LIN {X 0,Y 573.583,Z 173.358,A -85,B 0,C 180,E1 -2266.731,E2 -2266.731} C_VEL
LIN {X 0,Y 573.739,Z 153.891,A -85,B 0,C 180,E1 -2269.402,E2 -2269.402} C_VEL
LIN {X 0,Y 573.978,Z 134.192,A -85,B 0,C 180,E1 -2272.118,E2 -2272.118} C_VEL
LIN {X 0,Y 573.92,Z 125.746,A -85,B 0,C 180,E1 -2273.303,E2 -2273.303} C_VEL
LIN {X 0,Y 573.25,Z 122.082,A -85,B 0,C 180,E1 -2273.864,E2 -2273.864} C_VEL
LIN {X 0,Y 573.237,Z 122.08,A -85,B 0,C 180,E1 -2276.492,E2 -2276.492} C_VEL
LIN {X 0,Y 573.262,Z 122.073,A -85,B 0,C 180,E1 -2279.366,E2 -2279.366} C_VEL
LIN {X 0,Y 573.25,Z 122.079,A -85,B 0,C 180,E1 -2282.227,E2 -2282.227} C_VEL
LIN {X 0,Y 573.235,Z 122.075,A -85,B 0,C 180,E1 -2284.771,E2 -2284.771} C_VEL
LIN {X 0,Y 573.236,Z 122.084,A -85,B 0,C 180,E1 -2287.807,E2 -2287.807} C_VEL
LIN {X 0,Y 573.246,Z 122.074,A -85,B 0,C 180,E1 -2290.525,E2 -2290.525} C_VEL
LIN {X 0,Y 573.237,Z 122.078,A -85,B 0,C 180,E1 -2293.359,E2 -2293.359} C_VEL
LIN {X 0,Y 573.246,Z 122.075,A -85,B 0,C 180,E1 -2296.331,E2 -2296.331} C_VEL
LIN {X 0,Y 573.23,Z 122.075,A -85,B 0,C 180,E1 -2298.543,E2 -2298.543} C_VEL
LIN {X 0,Y 573.242,Z 122.079,A -85,B 0,C 180,E1 -2301.298,E2 -2301.298} C_VEL
LIN {X 0,Y 573.213,Z 122.08,A -85,B 0,C 180,E1 -2304.018,E2 -2304.018} C_VEL
LIN {X 0,Y 573.239,Z 122.074,A -85,B 0,C 180,E1 -2306.516,E2 -2306.516} C_VEL
LIN {X 0,Y 573.224,Z 122.081,A -85,B 0,C 180,E1 -2309.118,E2 -2309.118} C_VEL
LIN {X 0,Y 573.251,Z 122.074,A -85,B 0,C 180,E1 -2311.971,E2 -2311.971} C_VEL
LIN {X 0,Y 573.248,Z 122.074,A -85,B 0,C 180,E1 -2314.589,E2 -2314.589} C_VEL
LIN {X 0,Y 573.235,Z 122.078,A -85,B 0,C 180,E1 -2317.662,E2 -2317.662} C_VEL
LIN {X 0,Y 573.267,Z 122.074,A -85,B 0,C 180,E1 -2320.67,E2 -2320.67} C_VEL
LIN {X 0,Y 573.24,Z 122.076,A -85,B 0,C 180,E1 -2323.621,E2 -2323.621} C_VEL
LIN {X 0,Y 573.273,Z 122.07,A -85,B 0,C 180,E1 -2325.807,E2 -2325.807} C_VEL
LIN {X 0,Y 573.264,Z 122.078,A -85,B 0,C 180,E1 -2328.745,E2 -2328.745} C_VEL
LIN {X 0,Y 573.254,Z 122.073,A -85,B 0,C 180,E1 -2331.54,E2 -2331.54} C_VEL
LIN {X 0,Y 573.298,Z 122.07,A -85,B 0,C 180,E1 -2334.372,E2 -2334.372} C_VEL
LIN {X 0,Y 573.313,Z 122.065,A -85,B 0,C 180,E1 -2337.892,E2 -2337.892} C_VEL
LIN {X 0,Y 573.334,Z 122.072,A -85,B 0,C 180,E1 -2340.702,E2 -2340.702} C_VEL
LIN {X 0,Y 573.305,Z 122.073,A -85,B 0,C 180,E1 -2342.81,E2 -2342.81} C_VEL
LIN {X 0,Y 573.29,Z 122.068,A -85,B 0,C 180,E1 -2345.628,E2 -2345.628} C_VEL
LIN {X 0,Y 573.283,Z 122.078,A -85,B 0,C 180,E1 -2348.459,E2 -2348.459} C_VEL
LIN {X 0,Y 573.272,Z 122.07,A -85,B 0,C 180,E1 -2351.312,E2 -2351.312} C_VEL
LIN {X 0,Y 573.281,Z 122.078,A -85,B 0,C 180,E1 -2354.424,E2 -2354.424} C_VEL
LIN {X 0,Y 573.258,Z 122.072,A -85,B 0,C 180,E1 -2357.111,E2 -2357.111} C_VEL
LIN {X 0,Y 573.24,Z 122.081,A -85,B 0,C 180,E1 -2360.077,E2 -2360.077} C_VEL
LIN {X 0,Y 573.234,Z 122.082,A -85,B 0,C 180,E1 -2362.338,E2 -2362.338} C_VEL
LIN {X 0,Y 573.248,Z 122.075,A -85,B 0,C 180,E1 -2364.39,E2 -2364.39} C_VEL
LIN {X 0,Y 572.622,Z 122.155,A -85,B 0,C 180,E1 -2364.976,E2 -2364.976} C_VEL
LIN {X 0,Y 569.773,Z 122.513,A -85,B 0,C 180,E1 -2365.927,E2 -2365.927} C_VEL
LIN {X 0,Y 567.334,Z 122.813,A -85,B 0,C 180,E1 -2366.693,E2 -2366.693} C_VEL
LIN {X 0,Y 566.275,Z 122.942,A -85,B 0,C 180,E1 -2367.284,E2 -2367.284} C_VEL
LIN {X 0,Y 566.184,Z 122.954,A -85,B 0,C 180,E1 -2367.484,E2 -2367.484} C_VEL
LIN {X 0,Y 566.199,Z 122.957,A -85,B 0,C 180,E1 -2369.769,E2 -2369.769} C_VEL
LIN {X 0,Y 566.201,Z 122.954,A -85,B 0,C 180,E1 -2372.43,E2 -2372.43} C_VEL
LIN {X 0,Y 566.178,Z 122.954,A -85,B 0,C 180,E1 -2374.989,E2 -2374.989} C_VEL
LIN {X 0,Y 566.195,Z 122.956,A -85,B 0,C 180,E1 -2377.461,E2 -2377.461} C_VEL
LIN {X 0,Y 566.208,Z 122.953,A -85,B 0,C 180,E1 -2380.199,E2 -2380.199} C_VEL
LIN {X 0,Y 566.199,Z 122.952,A -85,B 0,C 180,E1 -2383.054,E2 -2383.054} C_VEL
LIN {X 0,Y 566.197,Z 122.955,A -85,B 0,C 180,E1 -2386.049,E2 -2386.049} C_VEL
LIN {X 0,Y 566.203,Z 122.955,A -85,B 0,C 180,E1 -2389.215,E2 -2389.215} C_VEL
LIN {X 0,Y 566.184,Z 122.961,A -85,B 0,C 180,E1 -2391.637,E2 -2391.637} C_VEL
LIN {X 0,Y 566.161,Z 122.956,A -85,B 0,C 180,E1 -2394.308,E2 -2394.308} C_VEL
LIN {X 0,Y 566.203,Z 122.953,A -85,B 0,C 180,E1 -2396.897,E2 -2396.897} C_VEL
LIN {X 0,Y 566.174,Z 122.963,A -85,B 0,C 180,E1 -2399.407,E2 -2399.407} C_VEL
LIN {X 0,Y 566.194,Z 122.954,A -85,B 0,C 180,E1 -2401.857,E2 -2401.857} C_VEL
LIN {X 0,Y 566.209,Z 122.95,A -85,B 0,C 180,E1 -2404.251,E2 -2404.251} C_VEL
LIN {X 0,Y 566.168,Z 122.958,A -85,B 0,C 180,E1 -2406.72,E2 -2406.72} C_VEL
LIN {X 0,Y 566.205,Z 122.952,A -85,B 0,C 180,E1 -2409.663,E2 -2409.663} C_VEL
LIN {X 0,Y 566.196,Z 122.956,A -85,B 0,C 180,E1 -2412.668,E2 -2412.668} C_VEL
LIN {X 0,Y 566.221,Z 122.95,A -85,B 0,C 180,E1 -2415.627,E2 -2415.627} C_VEL
LIN {X 0,Y 566.235,Z 122.953,A -85,B 0,C 180,E1 -2418.676,E2 -2418.676} C_VEL
LIN {X 0,Y 566.205,Z 122.952,A -85,B 0,C 180,E1 -2421.434,E2 -2421.434} C_VEL
LIN {X 0,Y 566.265,Z 122.946,A -85,B 0,C 180,E1 -2424.302,E2 -2424.302} C_VEL
LIN {X 0,Y 566.283,Z 122.942,A -85,B 0,C 180,E1 -2427.866,E2 -2427.866} C_VEL
LIN {X 0,Y 566.303,Z 122.948,A -85,B 0,C 180,E1 -2430.711,E2 -2430.711} C_VEL
LIN {X 0,Y 566.274,Z 123.08,A -85,B 0,C 180,E1 -2431.6,E2 -2431.6} C_VEL
LIN {X 0,Y 566.359,Z 131.56,A -85,B 0,C 180,E1 -2433.201,E2 -2433.201} C_VEL
LIN {X 0,Y 566.17,Z 146.716,A -85,B 0,C 180,E1 -2436.057,E2 -2436.057} C_VEL
LIN {X 0,Y 567.134,Z 152.715,A -85,B 0,C 180,E1 -2436.158,E2 -2436.158} C_VEL
LIN {X 0,Y 566.874,Z 253.461,A -85,B 0,C 180,E1 -2437.456,E2 -2437.456} C_VEL
LIN {X 0,Y 566.817,Z 267.103,A -85,B 0,C 180,E1 -2437.79,E2 -2437.79} C_VEL
LIN {X 0,Y 566.718,Z 279.633,A -85,B 0,C 180,E1 -2438.244,E2 -2438.244} C_VEL
LIN {X 0,Y 566.604,Z 291.505,A -85,B 0,C 180,E1 -2438.83,E2 -2438.83} C_VEL
LIN {X 0,Y 566.448,Z 302.94,A -85,B 0,C 180,E1 -2439.552,E2 -2439.552} C_VEL
LIN {X 0,Y 566.305,Z 313.27,A -85,B 0,C 180,E1 -2440.367,E2 -2440.367} C_VEL
LIN {X 0,Y 566.179,Z 322.76,A -85,B 0,C 180,E1 -2441.296,E2 -2441.296} C_VEL
LIN {X 0,Y 566.072,Z 331.625,A -85,B 0,C 180,E1 -2442.367,E2 -2442.367} C_VEL
LIN {X 0,Y 566.022,Z 338.925,A -85,B 0,C 180,E1 -2443.463,E2 -2443.463} C_VEL
LIN {X 0,Y 565.955,Z 345.411,A -85,B 0,C 180,E1 -2444.711,E2 -2444.711} C_VEL
LIN {X 0,Y 565.893,Z 349.972,A -85,B 0,C 180,E1 -2445.856,E2 -2445.856} C_VEL
LIN {X 0,Y 565.855,Z 353.302,A -85,B 0,C 180,E1 -2446.991,E2 -2446.991} C_VEL
LIN {X 0,Y 565.837,Z 355.482,A -85,B 0,C 180,E1 -2448.09,E2 -2448.09} C_VEL
LIN {X 0,Y 565.872,Z 356.753,A -85,B 0,C 180,E1 -2449.283,E2 -2449.283} C_VEL
LIN {X 0,Y 565.836,Z 356.938,A -85,B 0,C 180,E1 -2450.351,E2 -2450.351} C_VEL
LIN {X 0,Y 565.864,Z 356.337,A -85,B 0,C 180,E1 -2451.331,E2 -2451.331} C_VEL
LIN {X 0,Y 565.858,Z 354.318,A -85,B 0,C 180,E1 -2452.645,E2 -2452.645} C_VEL
LIN {X 0,Y 565.904,Z 351.363,A -85,B 0,C 180,E1 -2453.805,E2 -2453.805} C_VEL
LIN {X 0,Y 565.924,Z 347.174,A -85,B 0,C 180,E1 -2454.976,E2 -2454.976} C_VEL
LIN {X 0,Y 565.99,Z 341.588,A -85,B 0,C 180,E1 -2456.156,E2 -2456.156} C_VEL
LIN {X 0,Y 566.049,Z 334.295,A -85,B 0,C 180,E1 -2457.348,E2 -2457.348} C_VEL
LIN {X 0,Y 566.132,Z 326.85,A -85,B 0,C 180,E1 -2458.329,E2 -2458.329} C_VEL
LIN {X 0,Y 566.255,Z 317.253,A -85,B 0,C 180,E1 -2459.357,E2 -2459.357} C_VEL
LIN {X 0,Y 566.365,Z 306.538,A -85,B 0,C 180,E1 -2460.273,E2 -2460.273} C_VEL
LIN {X 0,Y 566.505,Z 295.04,A -85,B 0,C 180,E1 -2461.058,E2 -2461.058} C_VEL
LIN {X 0,Y 566.696,Z 282.783,A -85,B 0,C 180,E1 -2461.704,E2 -2461.704} C_VEL
LIN {X 0,Y 566.826,Z 269.71,A -85,B 0,C 180,E1 -2462.219,E2 -2462.219} C_VEL
LIN {X 0,Y 566.924,Z 256.913,A -85,B 0,C 180,E1 -2462.564,E2 -2462.564} C_VEL
LIN {X 0,Y 566.964,Z 241.389,A -85,B 0,C 180,E1 -2462.805,E2 -2462.805} C_VEL
LIN {X 0,Y 567.146,Z 152.118,A -85,B 0,C 180,E1 -2463.939,E2 -2463.939} C_VEL
LIN {X 0,Y 566.206,Z 146.617,A -85,B 0,C 180,E1 -2464.047,E2 -2464.047} C_VEL
LIN {X 0,Y 566.359,Z 132.186,A -85,B 0,C 180,E1 -2466.776,E2 -2466.776} C_VEL
LIN {X 0,Y 566.237,Z 123.074,A -85,B 0,C 180,E1 -2468.463,E2 -2468.463} C_VEL
LIN {X 0,Y 566.166,Z 122.963,A -85,B 0,C 180,E1 -2471.141,E2 -2471.141} C_VEL
LIN {X 0,Y 566.158,Z 122.959,A -85,B 0,C 180,E1 -2474.04,E2 -2474.04} C_VEL
LIN {X 0,Y 566.182,Z 122.963,A -85,B 0,C 180,E1 -2477.085,E2 -2477.085} C_VEL
LIN {X 0,Y 566.205,Z 122.952,A -85,B 0,C 180,E1 -2479.801,E2 -2479.801} C_VEL
LIN {X 0,Y 566.192,Z 122.956,A -85,B 0,C 180,E1 -2482.6,E2 -2482.6} C_VEL
LIN {X 0,Y 566.182,Z 122.96,A -85,B 0,C 180,E1 -2485.18,E2 -2485.18} C_VEL
LIN {X 0,Y 566.217,Z 122.95,A -85,B 0,C 180,E1 -2487.743,E2 -2487.743} C_VEL
LIN {X 0,Y 566.149,Z 122.961,A -85,B 0,C 180,E1 -2490.338,E2 -2490.338} C_VEL
LIN {X 0,Y 566.175,Z 122.956,A -85,B 0,C 180,E1 -2493.457,E2 -2493.457} C_VEL
LIN {X 0,Y 566.151,Z 122.958,A -85,B 0,C 180,E1 -2495.817,E2 -2495.817} C_VEL
LIN {X 0,Y 566.182,Z 122.958,A -85,B 0,C 180,E1 -2498.901,E2 -2498.901} C_VEL
LIN {X 0,Y 566.149,Z 122.959,A -85,B 0,C 180,E1 -2501.92,E2 -2501.92} C_VEL
LIN {X 0,Y 566.145,Z 122.959,A -85,B 0,C 180,E1 -2504.889,E2 -2504.889} C_VEL
LIN {X 0,Y 566.16,Z 122.96,A -85,B 0,C 180,E1 -2507.817,E2 -2507.817} C_VEL
LIN {X 0,Y 566.153,Z 122.962,A -85,B 0,C 180,E1 -2509.992,E2 -2509.992} C_VEL
LIN {X 0,Y 566.182,Z 122.953,A -85,B 0,C 180,E1 -2512.87,E2 -2512.87} C_VEL
LIN {X 0,Y 566.246,Z 122.945,A -85,B 0,C 180,E1 -2515.016,E2 -2515.016} C_VEL
LIN {X 0,Y 566.278,Z 122.95,A -85,B 0,C 180,E1 -2517.866,E2 -2517.866} C_VEL
LIN {X 0,Y 566.286,Z 122.948,A -85,B 0,C 180,E1 -2520,E2 -2520} C_VEL
LIN {X 0,Y 566.238,Z 122.945,A -85,B 0,C 180,E1 -2522.846,E2 -2522.846} C_VEL
LIN {X 0,Y 566.239,Z 122.956,A -85,B 0,C 180,E1 -2525.699,E2 -2525.699} C_VEL
LIN {X 0,Y 566.188,Z 122.952,A -85,B 0,C 180,E1 -2528.566,E2 -2528.566} C_VEL
LIN {X 0,Y 566.241,Z 122.955,A -85,B 0,C 180,E1 -2531.454,E2 -2531.454} C_VEL
LIN {X 0,Y 566.215,Z 122.949,A -85,B 0,C 180,E1 -2534.498,E2 -2534.498} C_VEL
LIN {X 0,Y 566.184,Z 122.961,A -85,B 0,C 180,E1 -2537.332,E2 -2537.332} C_VEL
LIN {X 0,Y 566.2,Z 122.956,A -85,B 0,C 180,E1 -2539.581,E2 -2539.581} C_VEL
LIN {X 0,Y 566.187,Z 122.952,A -85,B 0,C 180,E1 -2541.863,E2 -2541.863} C_VEL
LIN {X 0,Y 566.18,Z 122.962,A -85,B 0,C 180,E1 -2545.021,E2 -2545.021} C_VEL
LIN {X 0,Y 566.174,Z 122.959,A -85,B 0,C 180,E1 -2547.341,E2 -2547.341} C_VEL
LIN {X 0,Y 566.17,Z 122.955,A -85,B 0,C 180,E1 -2549.771,E2 -2549.771} C_VEL
LIN {X 0,Y 566.195,Z 122.955,A -85,B 0,C 180,E1 -2552.428,E2 -2552.428} C_VEL
LIN {X 0,Y 566.18,Z 122.961,A -85,B 0,C 180,E1 -2554.989,E2 -2554.989} C_VEL
LIN {X 0,Y 566.197,Z 122.952,A -85,B 0,C 180,E1 -2557.461,E2 -2557.461} C_VEL
LIN {X 0,Y 566.208,Z 122.954,A -85,B 0,C 180,E1 -2560.199,E2 -2560.199} C_VEL
LIN {X 0,Y 566.19,Z 122.955,A -85,B 0,C 180,E1 -2563.056,E2 -2563.056} C_VEL
LIN {X 0,Y 566.195,Z 122.956,A -85,B 0,C 180,E1 -2566.049,E2 -2566.049} C_VEL
LIN {X 0,Y 566.206,Z 122.952,A -85,B 0,C 180,E1 -2569.215,E2 -2569.215} C_VEL
LIN {X 0,Y 566.187,Z 122.955,A -85,B 0,C 180,E1 -2571.637,E2 -2571.637} C_VEL
LIN {X 0,Y 566.153,Z 122.965,A -85,B 0,C 180,E1 -2574.307,E2 -2574.307} C_VEL
LIN {X 0,Y 566.222,Z 122.95,A -85,B 0,C 180,E1 -2576.898,E2 -2576.898} C_VEL
LIN {X 0,Y 566.174,Z 122.957,A -85,B 0,C 180,E1 -2579.407,E2 -2579.407} C_VEL
LIN {X 0,Y 566.194,Z 122.961,A -85,B 0,C 180,E1 -2581.856,E2 -2581.856} C_VEL
LIN {X 0,Y 566.213,Z 122.956,A -85,B 0,C 180,E1 -2584.251,E2 -2584.251} C_VEL
LIN {X 0,Y 566.251,Z 123.143,A -85,B 0,C 180,E1 -2586.065,E2 -2586.065} C_VEL
LIN {X 0,Y 567.011,Z 128.298,A -85,B 0,C 180,E1 -2586.825,E2 -2586.825} C_VEL
LIN {X 0,Y 566.878,Z 144.645,A -85,B 0,C 180,E1 -2589.118,E2 -2589.118} C_VEL
LIN {X 0,Y 566.673,Z 166.374,A -85,B 0,C 180,E1 -2592.124,E2 -2592.124} C_VEL
LIN {X 0,Y 566.453,Z 186.626,A -85,B 0,C 180,E1 -2594.897,E2 -2594.897} C_VEL
LIN {X 0,Y 566.408,Z 194.521,A -85,B 0,C 180,E1 -2595.986,E2 -2595.986} C_VEL
LIN {X 0,Y 567.163,Z 201.229,A -85,B 0,C 180,E1 -2596.095,E2 -2596.095} C_VEL
LIN {X 0,Y 566.939,Z 302.939,A -85,B 0,C 180,E1 -2597.402,E2 -2597.402} C_VEL
LIN {X 0,Y 566.856,Z 316.212,A -85,B 0,C 180,E1 -2597.719,E2 -2597.719} C_VEL
LIN {X 0,Y 566.742,Z 328.374,A -85,B 0,C 180,E1 -2598.148,E2 -2598.148} C_VEL
LIN {X 0,Y 566.608,Z 340.191,A -85,B 0,C 180,E1 -2598.71,E2 -2598.71} C_VEL
LIN {X 0,Y 566.439,Z 352.194,A -85,B 0,C 180,E1 -2599.455,E2 -2599.455} C_VEL
LIN {X 0,Y 566.325,Z 362.603,A -85,B 0,C 180,E1 -2600.265,E2 -2600.265} C_VEL
LIN {X 0,Y 566.207,Z 371.112,A -85,B 0,C 180,E1 -2601.074,E2 -2601.074} C_VEL
LIN {X 0,Y 566.112,Z 378.959,A -85,B 0,C 180,E1 -2601.972,E2 -2601.972} C_VEL
LIN {X 0,Y 566.001,Z 386.622,A -85,B 0,C 180,E1 -2603.046,E2 -2603.046} C_VEL
LIN {X 0,Y 566.004,Z 393.679,A -85,B 0,C 180,E1 -2604.299,E2 -2604.299} C_VEL
LIN {X 0,Y 565.933,Z 398.372,A -85,B 0,C 180,E1 -2605.37,E2 -2605.37} C_VEL
LIN {X 0,Y 565.927,Z 401.958,A -85,B 0,C 180,E1 -2606.44,E2 -2606.44} C_VEL
LIN {X 0,Y 565.878,Z 403.807,A -85,B 0,C 180,E1 -2607.152,E2 -2607.152} C_VEL
LIN {X 0,Y 565.846,Z 406.184,A -85,B 0,C 180,E1 -2608.576,E2 -2608.576} C_VEL
LIN {X 0,Y 565.839,Z 407,A -85,B 0,C 180,E1 -2610,E2 -2610} C_VEL
LIN {X 0,Y 565.846,Z 406.185,A -85,B 0,C 180,E1 -2611.423,E2 -2611.423} C_VEL
LIN {X 0,Y 565.878,Z 403.81,A -85,B 0,C 180,E1 -2612.847,E2 -2612.847} C_VEL
LIN {X 0,Y 565.926,Z 400.896,A -85,B 0,C 180,E1 -2613.916,E2 -2613.916} C_VEL
LIN {X 0,Y 565.878,Z 396.949,A -85,B 0,C 180,E1 -2614.987,E2 -2614.987} C_VEL
LIN {X 0,Y 566.002,Z 391.868,A -85,B 0,C 180,E1 -2616.058,E2 -2616.058} C_VEL
LIN {X 0,Y 566.04,Z 385.468,A -85,B 0,C 180,E1 -2617.132,E2 -2617.132} C_VEL
LIN {X 0,Y 566.134,Z 377.479,A -85,B 0,C 180,E1 -2618.208,E2 -2618.208} C_VEL
LIN {X 0,Y 566.229,Z 369.335,A -85,B 0,C 180,E1 -2619.105,E2 -2619.105} C_VEL
LIN {X 0,Y 566.347,Z 359.4,A -85,B 0,C 180,E1 -2620.005,E2 -2620.005} C_VEL
LIN {X 0,Y 566.536,Z 348.293,A -85,B 0,C 180,E1 -2620.807,E2 -2620.807} C_VEL
LIN {X 0,Y 566.613,Z 337.175,A -85,B 0,C 180,E1 -2621.447,E2 -2621.447} C_VEL
LIN {X 0,Y 566.776,Z 324.981,A -85,B 0,C 180,E1 -2621.987,E2 -2621.987} C_VEL
LIN {X 0,Y 566.914,Z 312.179,A -85,B 0,C 180,E1 -2622.393,E2 -2622.393} C_VEL
LIN {X 0,Y 566.957,Z 298.608,A -85,B 0,C 180,E1 -2622.665,E2 -2622.665} C_VEL
LIN {X 0,Y 567.061,Z 198.935,A -85,B 0,C 180,E1 -2623.937,E2 -2623.937} C_VEL
LIN {X 0,Y 566.42,Z 194.439,A -85,B 0,C 180,E1 -2624.024,E2 -2624.024} C_VEL
LIN {X 0,Y 566.627,Z 171.851,A -85,B 0,C 180,E1 -2627.128,E2 -2627.128} C_VEL
LIN {X 0,Y 566.864,Z 150.169,A -85,B 0,C 180,E1 -2630.123,E2 -2630.123} C_VEL
LIN {X 0,Y 567.079,Z 129.824,A -85,B 0,C 180,E1 -2632.979,E2 -2632.979} C_VEL
LIN {X 0,Y 566.804,Z 125.892,A -85,B 0,C 180,E1 -2633.551,E2 -2633.551} C_VEL
LIN {X 0,Y 566.22,Z 122.959,A -85,B 0,C 180,E1 -2634.009,E2 -2634.009} C_VEL
LIN {X 0,Y 566.203,Z 122.954,A -85,B 0,C 180,E1 -2636.657,E2 -2636.657} C_VEL
LIN {X 0,Y 566.203,Z 122.956,A -85,B 0,C 180,E1 -2639.671,E2 -2639.671} C_VEL
LIN {X 0,Y 566.203,Z 122.954,A -85,B 0,C 180,E1 -2642.429,E2 -2642.429} C_VEL
LIN {X 0,Y 566.18,Z 122.954,A -85,B 0,C 180,E1 -2644.989,E2 -2644.989} C_VEL
LIN {X 0,Y 566.198,Z 122.955,A -85,B 0,C 180,E1 -2647.461,E2 -2647.461} C_VEL
LIN {X 0,Y 566.21,Z 122.954,A -85,B 0,C 180,E1 -2650.199,E2 -2650.199} C_VEL
LIN {X 0,Y 566.201,Z 122.952,A -85,B 0,C 180,E1 -2653.054,E2 -2653.054} C_VEL
LIN {X 0,Y 566.199,Z 122.955,A -85,B 0,C 180,E1 -2656.049,E2 -2656.049} C_VEL
LIN {X 0,Y 566.205,Z 122.954,A -85,B 0,C 180,E1 -2659.214,E2 -2659.214} C_VEL
LIN {X 0,Y 566.186,Z 122.962,A -85,B 0,C 180,E1 -2661.637,E2 -2661.637} C_VEL
LIN {X 0,Y 566.162,Z 122.956,A -85,B 0,C 180,E1 -2664.308,E2 -2664.308} C_VEL
LIN {X 0,Y 566.204,Z 122.953,A -85,B 0,C 180,E1 -2666.897,E2 -2666.897} C_VEL
LIN {X 0,Y 566.176,Z 122.964,A -85,B 0,C 180,E1 -2669.407,E2 -2669.407} C_VEL
LIN {X 0,Y 566.213,Z 122.952,A -85,B 0,C 180,E1 -2671.857,E2 -2671.857} C_VEL
LIN {X 0,Y 566.21,Z 122.95,A -85,B 0,C 180,E1 -2674.251,E2 -2674.251} C_VEL
LIN {X 0,Y 566.172,Z 122.957,A -85,B 0,C 180,E1 -2676.718,E2 -2676.718} C_VEL
LIN {X 0,Y 566.206,Z 122.953,A -85,B 0,C 180,E1 -2679.662,E2 -2679.662} C_VEL
LIN {X 0,Y 566.197,Z 122.955,A -85,B 0,C 180,E1 -2682.668,E2 -2682.668} C_VEL
LIN {X 0,Y 566.234,Z 122.948,A -85,B 0,C 180,E1 -2685.627,E2 -2685.627} C_VEL
LIN {X 0,Y 566.235,Z 122.952,A -85,B 0,C 180,E1 -2688.675,E2 -2688.675} C_VEL
LIN {X 0,Y 566.206,Z 122.952,A -85,B 0,C 180,E1 -2691.434,E2 -2691.434} C_VEL
LIN {X 0,Y 566.265,Z 122.945,A -85,B 0,C 180,E1 -2694.302,E2 -2694.302} C_VEL
LIN {X 0,Y 566.283,Z 122.941,A -85,B 0,C 180,E1 -2697.866,E2 -2697.866} C_VEL
LIN {X 0,Y 566.304,Z 122.948,A -85,B 0,C 180,E1 -2700.711,E2 -2700.711} C_VEL
LIN {X 0,Y 566.271,Z 122.948,A -85,B 0,C 180,E1 -2702.845,E2 -2702.845} C_VEL
LIN {X 0,Y 566.259,Z 122.944,A -85,B 0,C 180,E1 -2705.698,E2 -2705.698} C_VEL
LIN {X 0,Y 566.227,Z 122.957,A -85,B 0,C 180,E1 -2708.566,E2 -2708.566} C_VEL
LIN {X 0,Y 566.242,Z 122.946,A -85,B 0,C 180,E1 -2711.454,E2 -2711.454} C_VEL
LIN {X 0,Y 566.234,Z 122.954,A -85,B 0,C 180,E1 -2714.506,E2 -2714.506} C_VEL
LIN {X 0,Y 566.197,Z 122.951,A -85,B 0,C 180,E1 -2717.332,E2 -2717.332} C_VEL
LIN {X 0,Y 566.206,Z 122.958,A -85,B 0,C 180,E1 -2720.337,E2 -2720.337} C_VEL
LIN {X 0,Y 566.169,Z 122.955,A -85,B 0,C 180,E1 -2723.281,E2 -2723.281} C_VEL
LIN {X 0,Y 566.213,Z 122.954,A -85,B 0,C 180,E1 -2725.749,E2 -2725.749} C_VEL
LIN {X 0,Y 566.184,Z 122.954,A -85,B 0,C 180,E1 -2727.484,E2 -2727.484} C_VEL
LIN {X 0,Y 565.505,Z 123.047,A -85,B 0,C 180,E1 -2728.078,E2 -2728.078} C_VEL
LIN {X 0,Y 562.646,Z 123.4,A -85,B 0,C 180,E1 -2729.042,E2 -2729.042} C_VEL
LIN {X 0,Y 560.242,Z 123.7,A -85,B 0,C 180,E1 -2729.817,E2 -2729.817} C_VEL
LIN {X 0,Y 559.218,Z 123.825,A -85,B 0,C 180,E1 -2730.416,E2 -2730.416} C_VEL
LIN {X 0,Y 559.138,Z 123.832,A -85,B 0,C 180,E1 -2730.619,E2 -2730.619} C_VEL
LIN {X 0,Y 559.162,Z 123.832,A -85,B 0,C 180,E1 -2733.575,E2 -2733.575} C_VEL
LIN {X 0,Y 559.145,Z 123.832,A -85,B 0,C 180,E1 -2736.445,E2 -2736.445} C_VEL
LIN {X 0,Y 559.176,Z 123.826,A -85,B 0,C 180,E1 -2738.934,E2 -2738.934} C_VEL
LIN {X 0,Y 559.161,Z 123.837,A -85,B 0,C 180,E1 -2741.77,E2 -2741.77} C_VEL
LIN {X 0,Y 559.134,Z 123.831,A -85,B 0,C 180,E1 -2744.74,E2 -2744.74} C_VEL
LIN {X 0,Y 559.157,Z 123.833,A -85,B 0,C 180,E1 -2747.256,E2 -2747.256} C_VEL
LIN {X 0,Y 559.178,Z 123.827,A -85,B 0,C 180,E1 -2750.134,E2 -2750.134} C_VEL
LIN {X 0,Y 559.14,Z 123.832,A -85,B 0,C 180,E1 -2752.892,E2 -2752.892} C_VEL
LIN {X 0,Y 559.156,Z 123.83,A -85,B 0,C 180,E1 -2756.052,E2 -2756.052} C_VEL
LIN {X 0,Y 559.151,Z 123.833,A -85,B 0,C 180,E1 -2758.981,E2 -2758.981} C_VEL
LIN {X 0,Y 559.168,Z 123.832,A -85,B 0,C 180,E1 -2761.619,E2 -2761.619} C_VEL
LIN {X 0,Y 559.178,Z 123.827,A -85,B 0,C 180,E1 -2763.903,E2 -2763.903} C_VEL
LIN {X 0,Y 559.137,Z 123.833,A -85,B 0,C 180,E1 -2766.572,E2 -2766.572} C_VEL
LIN {X 0,Y 559.175,Z 123.831,A -85,B 0,C 180,E1 -2769.395,E2 -2769.395} C_VEL
LIN {X 0,Y 559.136,Z 123.832,A -85,B 0,C 180,E1 -2771.686,E2 -2771.686} C_VEL
LIN {X 0,Y 559.158,Z 123.828,A -85,B 0,C 180,E1 -2773.948,E2 -2773.948} C_VEL
LIN {X 0,Y 559.164,Z 123.828,A -85,B 0,C 180,E1 -2776.184,E2 -2776.184} C_VEL
LIN {X 0,Y 559.206,Z 123.827,A -85,B 0,C 180,E1 -2778.605,E2 -2778.605} C_VEL
LIN {X 0,Y 559.17,Z 123.829,A -85,B 0,C 180,E1 -2781.325,E2 -2781.325} C_VEL
LIN {X 0,Y 559.233,Z 123.821,A -85,B 0,C 180,E1 -2784.23,E2 -2784.23} C_VEL
LIN {X 0,Y 559.254,Z 123.818,A -85,B 0,C 180,E1 -2787.84,E2 -2787.84} C_VEL
LIN {X 0,Y 559.273,Z 123.824,A -85,B 0,C 180,E1 -2790.72,E2 -2790.72} C_VEL
LIN {X 0,Y 559.224,Z 124.003,A -85,B 0,C 180,E1 -2791.53,E2 -2791.53} C_VEL
LIN {X 0,Y 559.382,Z 131.087,A -85,B 0,C 180,E1 -2792.881,E2 -2792.881} C_VEL
LIN {X 0,Y 559.168,Z 146.822,A -85,B 0,C 180,E1 -2795.861,E2 -2795.861} C_VEL
LIN {X 0,Y 560.234,Z 153.136,A -85,B 0,C 180,E1 -2795.986,E2 -2795.986} C_VEL
LIN {X 0,Y 559.948,Z 253.755,A -85,B 0,C 180,E1 -2797.301,E2 -2797.301} C_VEL
LIN {X 0,Y 559.875,Z 267.311,A -85,B 0,C 180,E1 -2797.638,E2 -2797.638} C_VEL
LIN {X 0,Y 559.765,Z 279.239,A -85,B 0,C 180,E1 -2798.075,E2 -2798.075} C_VEL
LIN {X 0,Y 559.636,Z 291.207,A -85,B 0,C 180,E1 -2798.668,E2 -2798.668} C_VEL
LIN {X 0,Y 559.447,Z 302.668,A -85,B 0,C 180,E1 -2799.399,E2 -2799.399} C_VEL
LIN {X 0,Y 559.282,Z 313.04,A -85,B 0,C 180,E1 -2800.224,E2 -2800.224} C_VEL
LIN {X 0,Y 559.148,Z 321.458,A -85,B 0,C 180,E1 -2801.041,E2 -2801.041} C_VEL
LIN {X 0,Y 559.027,Z 330.783,A -85,B 0,C 180,E1 -2802.156,E2 -2802.156} C_VEL
LIN {X 0,Y 558.899,Z 338.248,A -85,B 0,C 180,E1 -2803.267,E2 -2803.267} C_VEL
LIN {X 0,Y 558.862,Z 344.601,A -85,B 0,C 180,E1 -2804.462,E2 -2804.462} C_VEL
LIN {X 0,Y 558.826,Z 349.574,A -85,B 0,C 180,E1 -2805.688,E2 -2805.688} C_VEL
LIN {X 0,Y 558.764,Z 353.61,A -85,B 0,C 180,E1 -2807.078,E2 -2807.078} C_VEL
LIN {X 0,Y 558.732,Z 355.876,A -85,B 0,C 180,E1 -2808.328,E2 -2808.328} C_VEL
LIN {X 0,Y 558.77,Z 356.824,A -85,B 0,C 180,E1 -2809.383,E2 -2809.383} C_VEL
LIN {X 0,Y 558.745,Z 356.873,A -85,B 0,C 180,E1 -2810.621,E2 -2810.621} C_VEL
LIN {X 0,Y 558.77,Z 356.224,A -85,B 0,C 180,E1 -2811.449,E2 -2811.449} C_VEL
LIN {X 0,Y 558.748,Z 355.253,A -85,B 0,C 180,E1 -2812.169,E2 -2812.169} C_VEL
LIN {X 0,Y 558.802,Z 352.777,A -85,B 0,C 180,E1 -2813.348,E2 -2813.348} C_VEL
LIN {X 0,Y 558.842,Z 349.17,A -85,B 0,C 180,E1 -2814.52,E2 -2814.52} C_VEL
LIN {X 0,Y 558.863,Z 344.209,A -85,B 0,C 180,E1 -2815.713,E2 -2815.713} C_VEL
LIN {X 0,Y 558.944,Z 337.682,A -85,B 0,C 180,E1 -2816.914,E2 -2816.914} C_VEL
LIN {X 0,Y 559.052,Z 329.444,A -85,B 0,C 180,E1 -2818.113,E2 -2818.113} C_VEL
LIN {X 0,Y 559.184,Z 320.514,A -85,B 0,C 180,E1 -2819.145,E2 -2819.145} C_VEL
LIN {X 0,Y 559.333,Z 310.509,A -85,B 0,C 180,E1 -2820.082,E2 -2820.082} C_VEL
LIN {X 0,Y 559.468,Z 299.782,A -85,B 0,C 180,E1 -2820.895,E2 -2820.895} C_VEL
LIN {X 0,Y 559.655,Z 288.926,A -85,B 0,C 180,E1 -2821.548,E2 -2821.548} C_VEL
LIN {X 0,Y 559.815,Z 276.18,A -85,B 0,C 180,E1 -2822.14,E2 -2822.14} C_VEL
LIN {X 0,Y 559.947,Z 263.306,A -85,B 0,C 180,E1 -2822.57,E2 -2822.57} C_VEL
LIN {X 0,Y 560.032,Z 250.014,A -85,B 0,C 180,E1 -2822.85,E2 -2822.85} C_VEL
LIN {X 0,Y 560.224,Z 152.75,A -85,B 0,C 180,E1 -2824.11,E2 -2824.11} C_VEL
LIN {X 0,Y 559.228,Z 146.882,A -85,B 0,C 180,E1 -2824.224,E2 -2824.224} C_VEL
LIN {X 0,Y 559.352,Z 133.557,A -85,B 0,C 180,E1 -2826.745,E2 -2826.745} C_VEL
LIN {X 0,Y 559.234,Z 124.092,A -85,B 0,C 180,E1 -2828.506,E2 -2828.506} C_VEL
LIN {X 0,Y 559.179,Z 123.832,A -85,B 0,C 180,E1 -2828.61,E2 -2828.61} C_VEL
LIN {X 0,Y 559.133,Z 123.838,A -85,B 0,C 180,E1 -2831.047,E2 -2831.047} C_VEL
LIN {X 0,Y 559.108,Z 123.84,A -85,B 0,C 180,E1 -2833.737,E2 -2833.737} C_VEL
LIN {X 0,Y 559.107,Z 123.837,A -85,B 0,C 180,E1 -2836.263,E2 -2836.263} C_VEL
LIN {X 0,Y 559.152,Z 123.838,A -85,B 0,C 180,E1 -2839.187,E2 -2839.187} C_VEL
LIN {X 0,Y 559.126,Z 123.833,A -85,B 0,C 180,E1 -2841.982,E2 -2841.982} C_VEL
LIN {X 0,Y 559.121,Z 123.839,A -85,B 0,C 180,E1 -2844.789,E2 -2844.789} C_VEL
LIN {X 0,Y 559.148,Z 123.834,A -85,B 0,C 180,E1 -2847.366,E2 -2847.366} C_VEL
LIN {X 0,Y 559.1,Z 123.838,A -85,B 0,C 180,E1 -2850.152,E2 -2850.152} C_VEL
LIN {X 0,Y 559.114,Z 123.837,A -85,B 0,C 180,E1 -2853.185,E2 -2853.185} C_VEL
LIN {X 0,Y 559.094,Z 123.837,A -85,B 0,C 180,E1 -2855.492,E2 -2855.492} C_VEL
LIN {X 0,Y 559.152,Z 123.838,A -85,B 0,C 180,E1 -2858.623,E2 -2858.623} C_VEL
LIN {X 0,Y 559.09,Z 123.837,A -85,B 0,C 180,E1 -2861.684,E2 -2861.684} C_VEL
LIN {X 0,Y 559.12,Z 123.837,A -85,B 0,C 180,E1 -2863.947,E2 -2863.947} C_VEL
LIN {X 0,Y 559.129,Z 123.839,A -85,B 0,C 180,E1 -2866.183,E2 -2866.183} C_VEL
LIN {X 0,Y 559.163,Z 123.826,A -85,B 0,C 180,E1 -2869.133,E2 -2869.133} C_VEL
LIN {X 0,Y 559.135,Z 123.84,A -85,B 0,C 180,E1 -2872.053,E2 -2872.053} C_VEL
LIN {X 0,Y 559.223,Z 123.82,A -85,B 0,C 180,E1 -2874.953,E2 -2874.953} C_VEL
LIN {X 0,Y 559.248,Z 123.825,A -85,B 0,C 180,E1 -2877.84,E2 -2877.84} C_VEL
LIN {X 0,Y 559.254,Z 123.824,A -85,B 0,C 180,E1 -2880,E2 -2880} C_VEL
LIN {X 0,Y 559.206,Z 123.821,A -85,B 0,C 180,E1 -2882.882,E2 -2882.882} C_VEL
LIN {X 0,Y 559.207,Z 123.831,A -85,B 0,C 180,E1 -2885.771,E2 -2885.771} C_VEL
LIN {X 0,Y 559.153,Z 123.828,A -85,B 0,C 180,E1 -2888.675,E2 -2888.675} C_VEL
LIN {X 0,Y 559.198,Z 123.831,A -85,B 0,C 180,E1 -2891.601,E2 -2891.601} C_VEL
LIN {X 0,Y 559.162,Z 123.828,A -85,B 0,C 180,E1 -2894.579,E2 -2894.579} C_VEL
LIN {X 0,Y 559.13,Z 123.837,A -85,B 0,C 180,E1 -2897.558,E2 -2897.558} C_VEL
LIN {X 0,Y 559.163,Z 123.83,A -85,B 0,C 180,E1 -2899.838,E2 -2899.838} C_VEL
LIN {X 0,Y 559.133,Z 123.83,A -85,B 0,C 180,E1 -2902.153,E2 -2902.153} C_VEL
LIN {X 0,Y 559.142,Z 123.838,A -85,B 0,C 180,E1 -2905.178,E2 -2905.178} C_VEL
LIN {X 0,Y 559.114,Z 123.835,A -85,B 0,C 180,E1 -2907.716,E2 -2907.716} C_VEL
LIN {X 0,Y 559.137,Z 123.831,A -85,B 0,C 180,E1 -2910.184,E2 -2910.184} C_VEL
LIN {X 0,Y 559.15,Z 123.837,A -85,B 0,C 180,E1 -2912.716,E2 -2912.716} C_VEL
LIN {X 0,Y 559.129,Z 123.835,A -85,B 0,C 180,E1 -2915.324,E2 -2915.324} C_VEL
LIN {X 0,Y 559.131,Z 123.833,A -85,B 0,C 180,E1 -2918.018,E2 -2918.018} C_VEL
LIN {X 0,Y 559.156,Z 123.836,A -85,B 0,C 180,E1 -2920.813,E2 -2920.813} C_VEL
LIN {X 0,Y 559.113,Z 123.835,A -85,B 0,C 180,E1 -2923.737,E2 -2923.737} C_VEL
LIN {X 0,Y 559.138,Z 123.838,A -85,B 0,C 180,E1 -2926.266,E2 -2926.266} C_VEL
LIN {X 0,Y 559.157,Z 123.83,A -85,B 0,C 180,E1 -2929.187,E2 -2929.187} C_VEL
LIN {X 0,Y 559.133,Z 123.838,A -85,B 0,C 180,E1 -2931.982,E2 -2931.982} C_VEL
LIN {X 0,Y 559.131,Z 123.833,A -85,B 0,C 180,E1 -2934.788,E2 -2934.788} C_VEL
LIN {X 0,Y 559.158,Z 123.831,A -85,B 0,C 180,E1 -2937.365,E2 -2937.365} C_VEL
LIN {X 0,Y 559.141,Z 123.839,A -85,B 0,C 180,E1 -2940.144,E2 -2940.144} C_VEL
LIN {X 0,Y 559.169,Z 123.83,A -85,B 0,C 180,E1 -2943.174,E2 -2943.174} C_VEL
LIN {X 0,Y 559.212,Z 123.976,A -85,B 0,C 180,E1 -2945.917,E2 -2945.917} C_VEL
LIN {X 0,Y 560.06,Z 129.466,A -85,B 0,C 180,E1 -2946.739,E2 -2946.739} C_VEL
LIN {X 0,Y 559.911,Z 145.656,A -85,B 0,C 180,E1 -2949.039,E2 -2949.039} C_VEL
LIN {X 0,Y 559.671,Z 167.384,A -85,B 0,C 180,E1 -2952.082,E2 -2952.082} C_VEL
LIN {X 0,Y 559.415,Z 187.685,A -85,B 0,C 180,E1 -2954.889,E2 -2954.889} C_VEL
LIN {X 0,Y 559.415,Z 194.271,A -85,B 0,C 180,E1 -2955.796,E2 -2955.796} C_VEL
LIN {X 0,Y 560.3,Z 202.134,A -85,B 0,C 180,E1 -2955.935,E2 -2955.935} C_VEL
LIN {X 0,Y 560.039,Z 302.937,A -85,B 0,C 180,E1 -2957.245,E2 -2957.245} C_VEL
LIN {X 0,Y 559.923,Z 316.212,A -85,B 0,C 180,E1 -2957.564,E2 -2957.564} C_VEL
LIN {X 0,Y 559.789,Z 328.373,A -85,B 0,C 180,E1 -2957.999,E2 -2957.999} C_VEL
LIN {X 0,Y 559.642,Z 339.866,A -85,B 0,C 180,E1 -2958.55,E2 -2958.55} C_VEL
LIN {X 0,Y 559.474,Z 350.9,A -85,B 0,C 180,E1 -2959.23,E2 -2959.23} C_VEL
LIN {X 0,Y 559.316,Z 361.534,A -85,B 0,C 180,E1 -2960.051,E2 -2960.051} C_VEL
LIN {X 0,Y 559.162,Z 371.112,A -85,B 0,C 180,E1 -2960.961,E2 -2960.961} C_VEL
LIN {X 0,Y 559.05,Z 378.959,A -85,B 0,C 180,E1 -2961.869,E2 -2961.869} C_VEL
LIN {X 0,Y 558.943,Z 386.622,A -85,B 0,C 180,E1 -2962.958,E2 -2962.958} C_VEL
LIN {X 0,Y 558.936,Z 393.679,A -85,B 0,C 180,E1 -2964.227,E2 -2964.227} C_VEL
LIN {X 0,Y 558.826,Z 398.372,A -85,B 0,C 180,E1 -2965.311,E2 -2965.311} C_VEL
LIN {X 0,Y 558.836,Z 401.958,A -85,B 0,C 180,E1 -2966.395,E2 -2966.395} C_VEL
LIN {X 0,Y 558.799,Z 403.807,A -85,B 0,C 180,E1 -2967.116,E2 -2967.116} C_VEL
LIN {X 0,Y 558.745,Z 406.183,A -85,B 0,C 180,E1 -2968.558,E2 -2968.558} C_VEL
LIN {X 0,Y 558.74,Z 407,A -85,B 0,C 180,E1 -2970,E2 -2970} C_VEL
LIN {X 0,Y 558.745,Z 406.184,A -85,B 0,C 180,E1 -2971.441,E2 -2971.441} C_VEL
LIN {X 0,Y 558.799,Z 403.81,A -85,B 0,C 180,E1 -2972.884,E2 -2972.884} C_VEL
LIN {X 0,Y 558.844,Z 400.896,A -85,B 0,C 180,E1 -2973.966,E2 -2973.966} C_VEL
LIN {X 0,Y 558.798,Z 396.949,A -85,B 0,C 180,E1 -2975.051,E2 -2975.051} C_VEL
LIN {X 0,Y 558.922,Z 391.868,A -85,B 0,C 180,E1 -2976.135,E2 -2976.135} C_VEL
LIN {X 0,Y 558.977,Z 385.467,A -85,B 0,C 180,E1 -2977.223,E2 -2977.223} C_VEL
LIN {X 0,Y 559.099,Z 377.478,A -85,B 0,C 180,E1 -2978.312,E2 -2978.312} C_VEL
LIN {X 0,Y 559.194,Z 369.334,A -85,B 0,C 180,E1 -2979.221,E2 -2979.221} C_VEL
LIN {X 0,Y 559.357,Z 359.399,A -85,B 0,C 180,E1 -2980.131,E2 -2980.131} C_VEL
LIN {X 0,Y 559.556,Z 348.399,A -85,B 0,C 180,E1 -2980.937,E2 -2980.937} C_VEL
LIN {X 0,Y 559.671,Z 336.459,A -85,B 0,C 180,E1 -2981.628,E2 -2981.628} C_VEL
LIN {X 0,Y 559.82,Z 324.979,A -85,B 0,C 180,E1 -2982.138,E2 -2982.138} C_VEL
LIN {X 0,Y 559.968,Z 312.178,A -85,B 0,C 180,E1 -2982.549,E2 -2982.549} C_VEL
LIN {X 0,Y 560.042,Z 298.598,A -85,B 0,C 180,E1 -2982.824,E2 -2982.824} C_VEL
LIN {X 0,Y 560.223,Z 200.152,A -85,B 0,C 180,E1 -2984.093,E2 -2984.093} C_VEL
LIN {X 0,Y 559.412,Z 194.292,A -85,B 0,C 180,E1 -2984.204,E2 -2984.204} C_VEL
LIN {X 0,Y 559.621,Z 172.311,A -85,B 0,C 180,E1 -2987.243,E2 -2987.243} C_VEL
LIN {X 0,Y 559.875,Z 151.22,A -85,B 0,C 180,E1 -2990.194,E2 -2990.194} C_VEL
LIN {X 0,Y 560.132,Z 130.948,A -85,B 0,C 180,E1 -2993.077,E2 -2993.077} C_VEL
LIN {X 0,Y 559.762,Z 126.82,A -85,B 0,C 180,E1 -2993.689,E2 -2993.689} C_VEL
LIN {X 0,Y 559.181,Z 123.836,A -85,B 0,C 180,E1 -2994.158,E2 -2994.158} C_VEL
LIN {X 0,Y 559.166,Z 123.829,A -85,B 0,C 180,E1 -2996.902,E2 -2996.902} C_VEL
LIN {X 0,Y 559.149,Z 123.837,A -85,B 0,C 180,E1 -2999.857,E2 -2999.857} C_VEL
LIN {X 0,Y 559.158,Z 123.829,A -85,B 0,C 180,E1 -3002.715,E2 -3002.715} C_VEL
LIN {X 0,Y 559.128,Z 123.834,A -85,B 0,C 180,E1 -3005.324,E2 -3005.324} C_VEL
LIN {X 0,Y 559.134,Z 123.839,A -85,B 0,C 180,E1 -3008.017,E2 -3008.017} C_VEL
LIN {X 0,Y 559.157,Z 123.828,A -85,B 0,C 180,E1 -3010.812,E2 -3010.812} C_VEL
LIN {X 0,Y 559.157,Z 123.838,A -85,B 0,C 180,E1 -3013.732,E2 -3013.732} C_VEL
LIN {X 0,Y 559.148,Z 123.83,A -85,B 0,C 180,E1 -3016.803,E2 -3016.803} C_VEL
LIN {X 0,Y 559.156,Z 123.832,A -85,B 0,C 180,E1 -3019.187,E2 -3019.187} C_VEL
LIN {X 0,Y 559.133,Z 123.835,A -85,B 0,C 180,E1 -3021.982,E2 -3021.982} C_VEL
LIN {X 0,Y 559.132,Z 123.832,A -85,B 0,C 180,E1 -3024.787,E2 -3024.787} C_VEL
LIN {X 0,Y 559.154,Z 123.838,A -85,B 0,C 180,E1 -3027.365,E2 -3027.365} C_VEL
LIN {X 0,Y 559.145,Z 123.83,A -85,B 0,C 180,E1 -3030.143,E2 -3030.143} C_VEL
LIN {X 0,Y 559.17,Z 123.833,A -85,B 0,C 180,E1 -3033.097,E2 -3033.097} C_VEL
LIN {X 0,Y 559.156,Z 123.834,A -85,B 0,C 180,E1 -3035.495,E2 -3035.495} C_VEL
LIN {X 0,Y 559.172,Z 123.829,A -85,B 0,C 180,E1 -3038.624,E2 -3038.624} C_VEL
LIN {X 0,Y 559.161,Z 123.835,A -85,B 0,C 180,E1 -3040.926,E2 -3040.926} C_VEL
LIN {X 0,Y 559.16,Z 123.828,A -85,B 0,C 180,E1 -3043.948,E2 -3043.948} C_VEL
LIN {X 0,Y 559.171,Z 123.827,A -85,B 0,C 180,E1 -3046.184,E2 -3046.184} C_VEL
LIN {X 0,Y 559.194,Z 123.83,A -85,B 0,C 180,E1 -3049.133,E2 -3049.133} C_VEL
LIN {X 0,Y 559.196,Z 123.824,A -85,B 0,C 180,E1 -3052.053,E2 -3052.053} C_VEL
LIN {X 0,Y 559.25,Z 123.824,A -85,B 0,C 180,E1 -3054.953,E2 -3054.953} C_VEL
LIN {X 0,Y 559.254,Z 123.816,A -85,B 0,C 180,E1 -3057.839,E2 -3057.839} C_VEL
LIN {X 0,Y 559.274,Z 123.823,A -85,B 0,C 180,E1 -3060.72,E2 -3060.72} C_VEL
LIN {X 0,Y 559.237,Z 123.824,A -85,B 0,C 180,E1 -3062.881,E2 -3062.881} C_VEL
LIN {X 0,Y 559.229,Z 123.82,A -85,B 0,C 180,E1 -3065.77,E2 -3065.77} C_VEL
LIN {X 0,Y 559.185,Z 123.832,A -85,B 0,C 180,E1 -3068.674,E2 -3068.674} C_VEL
LIN {X 0,Y 559.205,Z 123.823,A -85,B 0,C 180,E1 -3071.6,E2 -3071.6} C_VEL
LIN {X 0,Y 559.2,Z 123.829,A -85,B 0,C 180,E1 -3074.595,E2 -3074.595} C_VEL
LIN {X 0,Y 559.141,Z 123.831,A -85,B 0,C 180,E1 -3077.557,E2 -3077.557} C_VEL
LIN {X 0,Y 559.165,Z 123.831,A -85,B 0,C 180,E1 -3079.838,E2 -3079.838} C_VEL
LIN {X 0,Y 559.14,Z 123.84,A -85,B 0,C 180,E1 -3082.153,E2 -3082.153} C_VEL
LIN {X 0,Y 559.176,Z 123.826,A -85,B 0,C 180,E1 -3085.298,E2 -3085.298} C_VEL
LIN {X 0,Y 559.139,Z 123.835,A -85,B 0,C 180,E1 -3087.714,E2 -3087.714} C_VEL
LIN {X 0,Y 559.138,Z 123.832,A -85,B 0,C 180,E1 -3090.619,E2 -3090.619} C_VEL
LIN {X 0,Y 558.476,Z 123.914,A -85,B 0,C 180,E1 -3091.22,E2 -3091.22} C_VEL
LIN {X 0,Y 555.614,Z 124.276,A -85,B 0,C 180,E1 -3092.197,E2 -3092.197} C_VEL
LIN {X 0,Y 553.202,Z 124.573,A -85,B 0,C 180,E1 -3092.982,E2 -3092.982} C_VEL
LIN {X 0,Y 552.182,Z 124.702,A -85,B 0,C 180,E1 -3093.589,E2 -3093.589} C_VEL
LIN {X 0,Y 552.108,Z 124.71,A -85,B 0,C 180,E1 -3093.794,E2 -3093.794} C_VEL
LIN {X 0,Y 552.104,Z 124.707,A -85,B 0,C 180,E1 -3096.747,E2 -3096.747} C_VEL
LIN {X 0,Y 552.132,Z 124.709,A -85,B 0,C 180,E1 -3099.527,E2 -3099.527} C_VEL
LIN {X 0,Y 552.129,Z 124.705,A -85,B 0,C 180,E1 -3102.425,E2 -3102.425} C_VEL
LIN {X 0,Y 552.095,Z 124.716,A -85,B 0,C 180,E1 -3105.563,E2 -3105.563} C_VEL
LIN {X 0,Y 552.12,Z 124.705,A -85,B 0,C 180,E1 -3108.554,E2 -3108.554} C_VEL
LIN {X 0,Y 552.116,Z 124.714,A -85,B 0,C 180,E1 -3111.411,E2 -3111.411} C_VEL
LIN {X 0,Y 552.085,Z 124.71,A -85,B 0,C 180,E1 -3114.156,E2 -3114.156} C_VEL
LIN {X 0,Y 552.106,Z 124.709,A -85,B 0,C 180,E1 -3116.814,E2 -3116.814} C_VEL
LIN {X 0,Y 552.099,Z 124.717,A -85,B 0,C 180,E1 -3119.391,E2 -3119.391} C_VEL
LIN {X 0,Y 552.105,Z 124.708,A -85,B 0,C 180,E1 -3121.902,E2 -3121.902} C_VEL
LIN {X 0,Y 552.155,Z 124.703,A -85,B 0,C 180,E1 -3124.65,E2 -3124.65} C_VEL
LIN {X 0,Y 552.091,Z 124.712,A -85,B 0,C 180,E1 -3127.549,E2 -3127.549} C_VEL
LIN {X 0,Y 552.144,Z 124.703,A -85,B 0,C 180,E1 -3130.375,E2 -3130.375} C_VEL
LIN {X 0,Y 552.154,Z 124.71,A -85,B 0,C 180,E1 -3132.977,E2 -3132.977} C_VEL
LIN {X 0,Y 552.13,Z 124.704,A -85,B 0,C 180,E1 -3136.004,E2 -3136.004} C_VEL
LIN {X 0,Y 552.162,Z 124.708,A -85,B 0,C 180,E1 -3138.994,E2 -3138.994} C_VEL
LIN {X 0,Y 552.15,Z 124.701,A -85,B 0,C 180,E1 -3141.952,E2 -3141.952} C_VEL
LIN {X 0,Y 552.226,Z 124.701,A -85,B 0,C 180,E1 -3144.889,E2 -3144.889} C_VEL
LIN {X 0,Y 552.225,Z 124.694,A -85,B 0,C 180,E1 -3147.812,E2 -3147.812} C_VEL
LIN {X 0,Y 552.243,Z 124.7,A -85,B 0,C 180,E1 -3150.729,E2 -3150.729} C_VEL
LIN {X 0,Y 552.137,Z 124.821,A -85,B 0,C 180,E1 -3151.436,E2 -3151.436} C_VEL
LIN {X 0,Y 552.425,Z 130.64,A -85,B 0,C 180,E1 -3152.552,E2 -3152.552} C_VEL
LIN {X 0,Y 552.194,Z 147.111,A -85,B 0,C 180,E1 -3155.684,E2 -3155.684} C_VEL
LIN {X 0,Y 553.386,Z 155.189,A -85,B 0,C 180,E1 -3155.831,E2 -3155.831} C_VEL
LIN {X 0,Y 553.041,Z 254.055,A -85,B 0,C 180,E1 -3157.14,E2 -3157.14} C_VEL
LIN {X 0,Y 552.947,Z 267.696,A -85,B 0,C 180,E1 -3157.484,E2 -3157.484} C_VEL
LIN {X 0,Y 552.831,Z 280.092,A -85,B 0,C 180,E1 -3157.947,E2 -3157.947} C_VEL
LIN {X 0,Y 552.681,Z 291.139,A -85,B 0,C 180,E1 -3158.501,E2 -3158.501} C_VEL
LIN {X 0,Y 552.483,Z 302.666,A -85,B 0,C 180,E1 -3159.242,E2 -3159.242} C_VEL
LIN {X 0,Y 552.282,Z 313.065,A -85,B 0,C 180,E1 -3160.077,E2 -3160.077} C_VEL
LIN {X 0,Y 552.121,Z 322.416,A -85,B 0,C 180,E1 -3161.008,E2 -3161.008} C_VEL
LIN {X 0,Y 551.969,Z 331.475,A -85,B 0,C 180,E1 -3162.128,E2 -3162.128} C_VEL
LIN {X 0,Y 551.823,Z 338.798,A -85,B 0,C 180,E1 -3163.253,E2 -3163.253} C_VEL
LIN {X 0,Y 551.79,Z 345.296,A -85,B 0,C 180,E1 -3164.536,E2 -3164.536} C_VEL
LIN {X 0,Y 551.729,Z 350.474,A -85,B 0,C 180,E1 -3165.895,E2 -3165.895} C_VEL
LIN {X 0,Y 551.681,Z 353.903,A -85,B 0,C 180,E1 -3167.168,E2 -3167.168} C_VEL
LIN {X 0,Y 551.646,Z 356.169,A -85,B 0,C 180,E1 -3168.572,E2 -3168.572} C_VEL
LIN {X 0,Y 551.68,Z 356.884,A -85,B 0,C 180,E1 -3169.489,E2 -3169.489} C_VEL
LIN {X 0,Y 551.644,Z 356.703,A -85,B 0,C 180,E1 -3170.899,E2 -3170.899} C_VEL
LIN {X 0,Y 551.654,Z 355.987,A -85,B 0,C 180,E1 -3171.682,E2 -3171.682} C_VEL
LIN {X 0,Y 551.662,Z 354.798,A -85,B 0,C 180,E1 -3172.47,E2 -3172.47} C_VEL
LIN {X 0,Y 551.73,Z 352.538,A -85,B 0,C 180,E1 -3173.488,E2 -3173.488} C_VEL
LIN {X 0,Y 551.758,Z 348.16,A -85,B 0,C 180,E1 -3174.856,E2 -3174.856} C_VEL
LIN {X 0,Y 551.812,Z 342.902,A -85,B 0,C 180,E1 -3176.066,E2 -3176.066} C_VEL
LIN {X 0,Y 551.91,Z 336.087,A -85,B 0,C 180,E1 -3177.286,E2 -3177.286} C_VEL
LIN {X 0,Y 552.007,Z 328.778,A -85,B 0,C 180,E1 -3178.326,E2 -3178.326} C_VEL
LIN {X 0,Y 552.166,Z 319.975,A -85,B 0,C 180,E1 -3179.343,E2 -3179.343} C_VEL
LIN {X 0,Y 552.319,Z 310.079,A -85,B 0,C 180,E1 -3180.273,E2 -3180.273} C_VEL
LIN {X 0,Y 552.497,Z 300.443,A -85,B 0,C 180,E1 -3181.009,E2 -3181.009} C_VEL
LIN {X 0,Y 552.716,Z 289.479,A -85,B 0,C 180,E1 -3181.682,E2 -3181.682} C_VEL
LIN {X 0,Y 552.89,Z 277.092,A -85,B 0,C 180,E1 -3182.268,E2 -3182.268} C_VEL
LIN {X 0,Y 553.055,Z 264.06,A -85,B 0,C 180,E1 -3182.716,E2 -3182.716} C_VEL
LIN {X 0,Y 553.122,Z 250.585,A -85,B 0,C 180,E1 -3183.008,E2 -3183.008} C_VEL
LIN {X 0,Y 553.368,Z 153.717,A -85,B 0,C 180,E1 -3184.278,E2 -3184.278} C_VEL
LIN {X 0,Y 552.227,Z 147.135,A -85,B 0,C 180,E1 -3184.41,E2 -3184.41} C_VEL
LIN {X 0,Y 552.377,Z 132.511,A -85,B 0,C 180,E1 -3187.182,E2 -3187.182} C_VEL
LIN {X 0,Y 552.195,Z 125.021,A -85,B 0,C 180,E1 -3188.583,E2 -3188.583} C_VEL
LIN {X 0,Y 552.134,Z 124.71,A -85,B 0,C 180,E1 -3188.706,E2 -3188.706} C_VEL
LIN {X 0,Y 552.074,Z 124.72,A -85,B 0,C 180,E1 -3191.45,E2 -3191.45} C_VEL
LIN {X 0,Y 552.075,Z 124.714,A -85,B 0,C 180,E1 -3194.53,E2 -3194.53} C_VEL
LIN {X 0,Y 552.086,Z 124.715,A -85,B 0,C 180,E1 -3197.59,E2 -3197.59} C_VEL
LIN {X 0,Y 552.125,Z 124.706,A -85,B 0,C 180,E1 -3200.473,E2 -3200.473} C_VEL
LIN {X 0,Y 552.098,Z 124.712,A -85,B 0,C 180,E1 -3203.319,E2 -3203.319} C_VEL
LIN {X 0,Y 552.096,Z 124.709,A -85,B 0,C 180,E1 -3205.937,E2 -3205.937} C_VEL
LIN {X 0,Y 552.079,Z 124.716,A -85,B 0,C 180,E1 -3208.538,E2 -3208.538} C_VEL
LIN {X 0,Y 552.071,Z 124.713,A -85,B 0,C 180,E1 -3211.449,E2 -3211.449} C_VEL
LIN {X 0,Y 552.074,Z 124.716,A -85,B 0,C 180,E1 -3214.353,E2 -3214.353} C_VEL
LIN {X 0,Y 552.044,Z 124.721,A -85,B 0,C 180,E1 -3216.756,E2 -3216.756} C_VEL
LIN {X 0,Y 552.066,Z 124.714,A -85,B 0,C 180,E1 -3219.118,E2 -3219.118} C_VEL
LIN {X 0,Y 552.044,Z 124.714,A -85,B 0,C 180,E1 -3221.442,E2 -3221.442} C_VEL
LIN {X 0,Y 552.066,Z 124.714,A -85,B 0,C 180,E1 -3223.736,E2 -3223.736} C_VEL
LIN {X 0,Y 552.09,Z 124.713,A -85,B 0,C 180,E1 -3226.003,E2 -3226.003} C_VEL
LIN {X 0,Y 552.125,Z 124.703,A -85,B 0,C 180,E1 -3228.993,E2 -3228.993} C_VEL
LIN {X 0,Y 552.104,Z 124.714,A -85,B 0,C 180,E1 -3231.951,E2 -3231.951} C_VEL
LIN {X 0,Y 552.2,Z 124.695,A -85,B 0,C 180,E1 -3234.889,E2 -3234.889} C_VEL
LIN {X 0,Y 552.219,Z 124.7,A -85,B 0,C 180,E1 -3237.812,E2 -3237.812} C_VEL
LIN {X 0,Y 552.223,Z 124.7,A -85,B 0,C 180,E1 -3240,E2 -3240} C_VEL
LIN {X 0,Y 552.175,Z 124.696,A -85,B 0,C 180,E1 -3242.918,E2 -3242.918} C_VEL
LIN {X 0,Y 552.176,Z 124.705,A -85,B 0,C 180,E1 -3245.844,E2 -3245.844} C_VEL
LIN {X 0,Y 552.127,Z 124.704,A -85,B 0,C 180,E1 -3248.786,E2 -3248.786} C_VEL
LIN {X 0,Y 552.152,Z 124.705,A -85,B 0,C 180,E1 -3251.751,E2 -3251.751} C_VEL
LIN {X 0,Y 552.123,Z 124.706,A -85,B 0,C 180,E1 -3254.749,E2 -3254.749} C_VEL
LIN {X 0,Y 552.088,Z 124.711,A -85,B 0,C 180,E1 -3257.789,E2 -3257.789} C_VEL
LIN {X 0,Y 552.125,Z 124.705,A -85,B 0,C 180,E1 -3260.102,E2 -3260.102} C_VEL
LIN {X 0,Y 552.085,Z 124.708,A -85,B 0,C 180,E1 -3262.451,E2 -3262.451} C_VEL
LIN {X 0,Y 552.109,Z 124.707,A -85,B 0,C 180,E1 -3265.645,E2 -3265.645} C_VEL
LIN {X 0,Y 552.061,Z 124.713,A -85,B 0,C 180,E1 -3268.101,E2 -3268.101} C_VEL
LIN {X 0,Y 552.094,Z 124.712,A -85,B 0,C 180,E1 -3270.61,E2 -3270.61} C_VEL
LIN {X 0,Y 552.106,Z 124.711,A -85,B 0,C 180,E1 -3273.187,E2 -3273.187} C_VEL
LIN {X 0,Y 552.087,Z 124.71,A -85,B 0,C 180,E1 -3275.844,E2 -3275.844} C_VEL
LIN {X 0,Y 552.12,Z 124.709,A -85,B 0,C 180,E1 -3279.061,E2 -3279.061} C_VEL
LIN {X 0,Y 552.112,Z 124.707,A -85,B 0,C 180,E1 -3281.447,E2 -3281.447} C_VEL
LIN {X 0,Y 552.078,Z 124.72,A -85,B 0,C 180,E1 -3284.53,E2 -3284.53} C_VEL
LIN {X 0,Y 552.111,Z 124.708,A -85,B 0,C 180,E1 -3287.587,E2 -3287.587} C_VEL
LIN {X 0,Y 552.135,Z 124.711,A -85,B 0,C 180,E1 -3290.473,E2 -3290.473} C_VEL
LIN {X 0,Y 552.102,Z 124.708,A -85,B 0,C 180,E1 -3293.318,E2 -3293.318} C_VEL
LIN {X 0,Y 552.128,Z 124.71,A -85,B 0,C 180,E1 -3295.939,E2 -3295.939} C_VEL
LIN {X 0,Y 552.123,Z 124.709,A -85,B 0,C 180,E1 -3298.541,E2 -3298.541} C_VEL
LIN {X 0,Y 552.105,Z 124.711,A -85,B 0,C 180,E1 -3301.442,E2 -3301.442} C_VEL
LIN {X 0,Y 552.132,Z 124.71,A -85,B 0,C 180,E1 -3304.356,E2 -3304.356} C_VEL
LIN {X 0,Y 552.155,Z 124.81,A -85,B 0,C 180,E1 -3305.764,E2 -3305.764} C_VEL
LIN {X 0,Y 553.163,Z 131.688,A -85,B 0,C 180,E1 -3306.805,E2 -3306.805} C_VEL
LIN {X 0,Y 552.916,Z 149.387,A -85,B 0,C 180,E1 -3309.346,E2 -3309.346} C_VEL
LIN {X 0,Y 552.604,Z 171.861,A -85,B 0,C 180,E1 -3312.526,E2 -3312.526} C_VEL
LIN {X 0,Y 552.371,Z 194.033,A -85,B 0,C 180,E1 -3315.626,E2 -3315.626} C_VEL
LIN {X 0,Y 553.425,Z 202.207,A -85,B 0,C 180,E1 -3315.762,E2 -3315.762} C_VEL
LIN {X 0,Y 553.106,Z 302.54,A -85,B 0,C 180,E1 -3317.082,E2 -3317.082} C_VEL
LIN {X 0,Y 552.966,Z 315.866,A -85,B 0,C 180,E1 -3317.405,E2 -3317.405} C_VEL
LIN {X 0,Y 552.819,Z 328.071,A -85,B 0,C 180,E1 -3317.845,E2 -3317.845} C_VEL
LIN {X 0,Y 552.638,Z 339.63,A -85,B 0,C 180,E1 -3318.402,E2 -3318.402} C_VEL
LIN {X 0,Y 552.481,Z 350.726,A -85,B 0,C 180,E1 -3319.092,E2 -3319.092} C_VEL
LIN {X 0,Y 552.298,Z 361.428,A -85,B 0,C 180,E1 -3319.923,E2 -3319.923} C_VEL
LIN {X 0,Y 552.131,Z 371.073,A -85,B 0,C 180,E1 -3320.845,E2 -3320.845} C_VEL
LIN {X 0,Y 552.013,Z 378.959,A -85,B 0,C 180,E1 -3321.765,E2 -3321.765} C_VEL
LIN {X 0,Y 551.889,Z 386.62,A -85,B 0,C 180,E1 -3322.868,E2 -3322.868} C_VEL
LIN {X 0,Y 551.867,Z 393.679,A -85,B 0,C 180,E1 -3324.152,E2 -3324.152} C_VEL
LIN {X 0,Y 551.725,Z 398.372,A -85,B 0,C 180,E1 -3325.25,E2 -3325.25} C_VEL
LIN {X 0,Y 551.75,Z 401.957,A -85,B 0,C 180,E1 -3326.348,E2 -3326.348} C_VEL
LIN {X 0,Y 551.724,Z 403.806,A -85,B 0,C 180,E1 -3327.079,E2 -3327.079} C_VEL
LIN {X 0,Y 551.645,Z 406.182,A -85,B 0,C 180,E1 -3328.54,E2 -3328.54} C_VEL
LIN {X 0,Y 551.64,Z 407,A -85,B 0,C 180,E1 -3330,E2 -3330} C_VEL
LIN {X 0,Y 551.645,Z 406.184,A -85,B 0,C 180,E1 -3331.46,E2 -3331.46} C_VEL
LIN {X 0,Y 551.723,Z 403.81,A -85,B 0,C 180,E1 -3332.921,E2 -3332.921} C_VEL
LIN {X 0,Y 551.764,Z 400.896,A -85,B 0,C 180,E1 -3334.017,E2 -3334.017} C_VEL
LIN {X 0,Y 551.723,Z 396.948,A -85,B 0,C 180,E1 -3335.116,E2 -3335.116} C_VEL
LIN {X 0,Y 551.803,Z 391.189,A -85,B 0,C 180,E1 -3336.341,E2 -3336.341} C_VEL
LIN {X 0,Y 551.926,Z 384.236,A -85,B 0,C 180,E1 -3337.499,E2 -3337.499} C_VEL
LIN {X 0,Y 552.082,Z 375.987,A -85,B 0,C 180,E1 -3338.602,E2 -3338.602} C_VEL
LIN {X 0,Y 552.2,Z 367.479,A -85,B 0,C 180,E1 -3339.523,E2 -3339.523} C_VEL
LIN {X 0,Y 552.412,Z 356.964,A -85,B 0,C 180,E1 -3340.445,E2 -3340.445} C_VEL
LIN {X 0,Y 552.555,Z 346.097,A -85,B 0,C 180,E1 -3341.214,E2 -3341.214} C_VEL
LIN {X 0,Y 552.752,Z 335.163,A -85,B 0,C 180,E1 -3341.831,E2 -3341.831} C_VEL
LIN {X 0,Y 552.9,Z 323.469,A -85,B 0,C 180,E1 -3342.34,E2 -3342.34} C_VEL
LIN {X 0,Y 553.052,Z 310.917,A -85,B 0,C 180,E1 -3342.732,E2 -3342.732} C_VEL
LIN {X 0,Y 553.127,Z 298.204,A -85,B 0,C 180,E1 -3342.987,E2 -3342.987} C_VEL
LIN {X 0,Y 553.243,Z 200.276,A -85,B 0,C 180,E1 -3344.268,E2 -3344.268} C_VEL
LIN {X 0,Y 552.383,Z 193.965,A -85,B 0,C 180,E1 -3344.392,E2 -3344.392} C_VEL
LIN {X 0,Y 552.603,Z 173.637,A -85,B 0,C 180,E1 -3347.239,E2 -3347.239} C_VEL
LIN {X 0,Y 552.899,Z 152.272,A -85,B 0,C 180,E1 -3350.266,E2 -3350.266} C_VEL
LIN {X 0,Y 553.212,Z 133.316,A -85,B 0,C 180,E1 -3352.995,E2 -3352.995} C_VEL
LIN {X 0,Y 552.839,Z 128.257,A -85,B 0,C 180,E1 -3353.75,E2 -3353.75} C_VEL
LIN {X 0,Y 552.12,Z 124.714,A -85,B 0,C 180,E1 -3354.337,E2 -3354.337} C_VEL
LIN {X 0,Y 552.136,Z 124.705,A -85,B 0,C 180,E1 -3356.999,E2 -3356.999} C_VEL
LIN {X 0,Y 552.118,Z 124.715,A -85,B 0,C 180,E1 -3360.05,E2 -3360.05} C_VEL
LIN {X 0,Y 552.116,Z 124.706,A -85,B 0,C 180,E1 -3362.846,E2 -3362.846} C_VEL
LIN {X 0,Y 552.078,Z 124.713,A -85,B 0,C 180,E1 -3365.439,E2 -3365.439} C_VEL
LIN {X 0,Y 552.098,Z 124.718,A -85,B 0,C 180,E1 -3367.885,E2 -3367.885} C_VEL
LIN {X 0,Y 552.111,Z 124.707,A -85,B 0,C 180,E1 -3370.481,E2 -3370.481} C_VEL
LIN {X 0,Y 552.121,Z 124.71,A -85,B 0,C 180,E1 -3373.484,E2 -3373.484} C_VEL
LIN {X 0,Y 552.108,Z 124.707,A -85,B 0,C 180,E1 -3376.576,E2 -3376.576} C_VEL
LIN {X 0,Y 552.109,Z 124.715,A -85,B 0,C 180,E1 -3379.519,E2 -3379.519} C_VEL
LIN {X 0,Y 552.093,Z 124.709,A -85,B 0,C 180,E1 -3382.336,E2 -3382.336} C_VEL
LIN {X 0,Y 552.083,Z 124.713,A -85,B 0,C 180,E1 -3385.051,E2 -3385.051} C_VEL
LIN {X 0,Y 552.115,Z 124.711,A -85,B 0,C 180,E1 -3387.681,E2 -3387.681} C_VEL
LIN {X 0,Y 552.108,Z 124.707,A -85,B 0,C 180,E1 -3390.235,E2 -3390.235} C_VEL
LIN {X 0,Y 552.139,Z 124.708,A -85,B 0,C 180,E1 -3393,E2 -3393} C_VEL
LIN {X 0,Y 552.114,Z 124.714,A -85,B 0,C 180,E1 -3395.161,E2 -3395.161} C_VEL
LIN {X 0,Y 552.126,Z 124.704,A -85,B 0,C 180,E1 -3398.337,E2 -3398.337} C_VEL
LIN {X 0,Y 552.151,Z 124.704,A -85,B 0,C 180,E1 -3400.674,E2 -3400.674} C_VEL
LIN {X 0,Y 552.111,Z 124.707,A -85,B 0,C 180,E1 -3403.737,E2 -3403.737} C_VEL
LIN {X 0,Y 552.135,Z 124.703,A -85,B 0,C 180,E1 -3406.004,E2 -3406.004} C_VEL
LIN {X 0,Y 552.162,Z 124.709,A -85,B 0,C 180,E1 -3408.993,E2 -3408.993} C_VEL
LIN {X 0,Y 552.15,Z 124.701,A -85,B 0,C 180,E1 -3411.951,E2 -3411.951} C_VEL
LIN {X 0,Y 552.226,Z 124.7,A -85,B 0,C 180,E1 -3414.889,E2 -3414.889} C_VEL
LIN {X 0,Y 552.225,Z 124.692,A -85,B 0,C 180,E1 -3417.812,E2 -3417.812} C_VEL
LIN {X 0,Y 552.243,Z 124.699,A -85,B 0,C 180,E1 -3420.729,E2 -3420.729} C_VEL
LIN {X 0,Y 552.203,Z 124.7,A -85,B 0,C 180,E1 -3422.918,E2 -3422.918} C_VEL
LIN {X 0,Y 552.199,Z 124.696,A -85,B 0,C 180,E1 -3425.844,E2 -3425.844} C_VEL
LIN {X 0,Y 552.153,Z 124.706,A -85,B 0,C 180,E1 -3428.786,E2 -3428.786} C_VEL
LIN {X 0,Y 552.162,Z 124.701,A -85,B 0,C 180,E1 -3431.75,E2 -3431.75} C_VEL
LIN {X 0,Y 552.136,Z 124.707,A -85,B 0,C 180,E1 -3434.748,E2 -3434.748} C_VEL
LIN {X 0,Y 552.098,Z 124.71,A -85,B 0,C 180,E1 -3437.789,E2 -3437.789} C_VEL
LIN {X 0,Y 552.126,Z 124.712,A -85,B 0,C 180,E1 -3440.101,E2 -3440.101} C_VEL
LIN {X 0,Y 552.091,Z 124.714,A -85,B 0,C 180,E1 -3442.451,E2 -3442.451} C_VEL
LIN {X 0,Y 552.155,Z 124.701,A -85,B 0,C 180,E1 -3445.35,E2 -3445.35} C_VEL
LIN {X 0,Y 552.089,Z 124.718,A -85,B 0,C 180,E1 -3448.099,E2 -3448.099} C_VEL
LIN {X 0,Y 552.101,Z 124.709,A -85,B 0,C 180,E1 -3450.615,E2 -3450.615} C_VEL
LIN {X 0,Y 552.114,Z 124.706,A -85,B 0,C 180,E1 -3453.186,E2 -3453.186} C_VEL
LIN {X 0,Y 552.108,Z 124.71,A -85,B 0,C 180,E1 -3453.794,E2 -3453.794} C_VEL
LIN {X 0,Y 551.474,Z 124.793,A -85,B 0,C 180,E1 -3454.403,E2 -3454.403} C_VEL
LIN {X 0,Y 548.651,Z 125.143,A -85,B 0,C 180,E1 -3455.391,E2 -3455.391} C_VEL
LIN {X 0,Y 546.23,Z 125.443,A -85,B 0,C 180,E1 -3456.186,E2 -3456.186} C_VEL
LIN {X 0,Y 545.161,Z 125.572,A -85,B 0,C 180,E1 -3456.8,E2 -3456.8} C_VEL
LIN {X 0,Y 545.06,Z 125.585,A -85,B 0,C 180,E1 -3457.008,E2 -3457.008} C_VEL
LIN {X 0,Y 545.067,Z 125.588,A -85,B 0,C 180,E1 -3460.142,E2 -3460.142} C_VEL
LIN {X 0,Y 545.077,Z 125.584,A -85,B 0,C 180,E1 -3463.107,E2 -3463.107} C_VEL
LIN {X 0,Y 545.066,Z 125.585,A -85,B 0,C 180,E1 -3466.224,E2 -3466.224} C_VEL
LIN {X 0,Y 545.08,Z 125.583,A -85,B 0,C 180,E1 -3468.885,E2 -3468.885} C_VEL
LIN {X 0,Y 545.079,Z 125.583,A -85,B 0,C 180,E1 -3470.818,E2 -3470.818} C_VEL
LIN {X 0,Y 545.041,Z 125.594,A -85,B 0,C 180,E1 -3473.62,E2 -3473.62} C_VEL
LIN {X 0,Y 545.049,Z 125.586,A -85,B 0,C 180,E1 -3476.327,E2 -3476.327} C_VEL
LIN {X 0,Y 545.064,Z 125.588,A -85,B 0,C 180,E1 -3478.952,E2 -3478.952} C_VEL
LIN {X 0,Y 545.1,Z 125.586,A -85,B 0,C 180,E1 -3481.508,E2 -3481.508} C_VEL
LIN {X 0,Y 545.094,Z 125.581,A -85,B 0,C 180,E1 -3484.492,E2 -3484.492} C_VEL
LIN {X 0,Y 545.036,Z 125.596,A -85,B 0,C 180,E1 -3487.242,E2 -3487.242} C_VEL
LIN {X 0,Y 545.116,Z 125.579,A -85,B 0,C 180,E1 -3490.415,E2 -3490.415} C_VEL
LIN {X 0,Y 545.067,Z 125.586,A -85,B 0,C 180,E1 -3493.521,E2 -3493.521} C_VEL
LIN {X 0,Y 545.09,Z 125.581,A -85,B 0,C 180,E1 -3495.82,E2 -3495.82} C_VEL
LIN {X 0,Y 545.118,Z 125.586,A -85,B 0,C 180,E1 -3498.849,E2 -3498.849} C_VEL
LIN {X 0,Y 545.098,Z 125.58,A -85,B 0,C 180,E1 -3501.847,E2 -3501.847} C_VEL
LIN {X 0,Y 545.202,Z 125.576,A -85,B 0,C 180,E1 -3504.823,E2 -3504.823} C_VEL
LIN {X 0,Y 545.196,Z 125.569,A -85,B 0,C 180,E1 -3507.784,E2 -3507.784} C_VEL
LIN {X 0,Y 545.212,Z 125.575,A -85,B 0,C 180,E1 -3510.739,E2 -3510.739} C_VEL
LIN {X 0,Y 545.109,Z 125.681,A -85,B 0,C 180,E1 -3511.339,E2 -3511.339} C_VEL
LIN {X 0,Y 545.421,Z 132.133,A -85,B 0,C 180,E1 -3512.585,E2 -3512.585} C_VEL
LIN {X 0,Y 545.212,Z 147.407,A -85,B 0,C 180,E1 -3515.502,E2 -3515.502} C_VEL
LIN {X 0,Y 546.513,Z 155.585,A -85,B 0,C 180,E1 -3515.65,E2 -3515.65} C_VEL
LIN {X 0,Y 546.167,Z 253.587,A -85,B 0,C 180,E1 -3516.96,E2 -3516.96} C_VEL
LIN {X 0,Y 546.046,Z 267.005,A -85,B 0,C 180,E1 -3517.292,E2 -3517.292} C_VEL
LIN {X 0,Y 545.892,Z 280.21,A -85,B 0,C 180,E1 -3517.783,E2 -3517.783} C_VEL
LIN {X 0,Y 545.758,Z 291.053,A -85,B 0,C 180,E1 -3518.33,E2 -3518.33} C_VEL
LIN {X 0,Y 545.52,Z 302.664,A -85,B 0,C 180,E1 -3519.08,E2 -3519.08} C_VEL
LIN {X 0,Y 545.304,Z 313.116,A -85,B 0,C 180,E1 -3519.926,E2 -3519.926} C_VEL
LIN {X 0,Y 545.118,Z 321.676,A -85,B 0,C 180,E1 -3520.775,E2 -3520.775} C_VEL
LIN {X 0,Y 545.015,Z 329.876,A -85,B 0,C 180,E1 -3521.761,E2 -3521.761} C_VEL
LIN {X 0,Y 544.854,Z 337.269,A -85,B 0,C 180,E1 -3522.856,E2 -3522.856} C_VEL
LIN {X 0,Y 544.77,Z 342.546,A -85,B 0,C 180,E1 -3523.808,E2 -3523.808} C_VEL
LIN {X 0,Y 544.725,Z 347.644,A -85,B 0,C 180,E1 -3524.954,E2 -3524.954} C_VEL
LIN {X 0,Y 544.626,Z 351.594,A -85,B 0,C 180,E1 -3526.108,E2 -3526.108} C_VEL
LIN {X 0,Y 544.582,Z 354.463,A -85,B 0,C 180,E1 -3527.267,E2 -3527.267} C_VEL
LIN {X 0,Y 544.568,Z 355.806,A -85,B 0,C 180,E1 -3528.043,E2 -3528.043} C_VEL
LIN {X 0,Y 544.582,Z 356.731,A -85,B 0,C 180,E1 -3528.822,E2 -3528.822} C_VEL
LIN {X 0,Y 544.576,Z 357.18,A -85,B 0,C 180,E1 -3529.606,E2 -3529.606} C_VEL
LIN {X 0,Y 544.567,Z 357.2,A -85,B 0,C 180,E1 -3530.393,E2 -3530.393} C_VEL
LIN {X 0,Y 544.571,Z 356.281,A -85,B 0,C 180,E1 -3531.69,E2 -3531.69} C_VEL
LIN {X 0,Y 544.58,Z 354.551,A -85,B 0,C 180,E1 -3532.778,E2 -3532.778} C_VEL
LIN {X 0,Y 544.658,Z 351.597,A -85,B 0,C 180,E1 -3533.982,E2 -3533.982} C_VEL
LIN {X 0,Y 544.692,Z 347.412,A -85,B 0,C 180,E1 -3535.201,E2 -3535.201} C_VEL
LIN {X 0,Y 544.808,Z 341.821,A -85,B 0,C 180,E1 -3536.427,E2 -3536.427} C_VEL
LIN {X 0,Y 544.914,Z 334.541,A -85,B 0,C 180,E1 -3537.666,E2 -3537.666} C_VEL
LIN {X 0,Y 545.06,Z 326.068,A -85,B 0,C 180,E1 -3538.815,E2 -3538.815} C_VEL
LIN {X 0,Y 545.237,Z 316.38,A -85,B 0,C 180,E1 -3539.859,E2 -3539.859} C_VEL
LIN {X 0,Y 545.406,Z 306.567,A -85,B 0,C 180,E1 -3540.718,E2 -3540.718} C_VEL
LIN {X 0,Y 545.606,Z 296.327,A -85,B 0,C 180,E1 -3541.445,E2 -3541.445} C_VEL
LIN {X 0,Y 545.876,Z 285.075,A -85,B 0,C 180,E1 -3542.079,E2 -3542.079} C_VEL
LIN {X 0,Y 546.051,Z 272.529,A -85,B 0,C 180,E1 -3542.613,E2 -3542.613} C_VEL
LIN {X 0,Y 546.2,Z 260.159,A -85,B 0,C 180,E1 -3542.986,E2 -3542.986} C_VEL
LIN {X 0,Y 546.285,Z 247.296,A -85,B 0,C 180,E1 -3543.227,E2 -3543.227} C_VEL
LIN {X 0,Y 546.527,Z 154.66,A -85,B 0,C 180,E1 -3544.452,E2 -3544.452} C_VEL
LIN {X 0,Y 545.232,Z 147.415,A -85,B 0,C 180,E1 -3544.594,E2 -3544.594} C_VEL
LIN {X 0,Y 545.367,Z 133.258,A -85,B 0,C 180,E1 -3547.278,E2 -3547.278} C_VEL
LIN {X 0,Y 545.28,Z 127.02,A -85,B 0,C 180,E1 -3548.454,E2 -3548.454} C_VEL
LIN {X 0,Y 545.115,Z 125.585,A -85,B 0,C 180,E1 -3548.763,E2 -3548.763} C_VEL
LIN {X 0,Y 545.039,Z 125.595,A -85,B 0,C 180,E1 -3551.593,E2 -3551.593} C_VEL
LIN {X 0,Y 545.038,Z 125.59,A -85,B 0,C 180,E1 -3554.131,E2 -3554.131} C_VEL
LIN {X 0,Y 545.017,Z 125.597,A -85,B 0,C 180,E1 -3556.887,E2 -3556.887} C_VEL
LIN {X 0,Y 545.062,Z 125.585,A -85,B 0,C 180,E1 -3559.857,E2 -3559.857} C_VEL
LIN {X 0,Y 545.064,Z 125.591,A -85,B 0,C 180,E1 -3563.075,E2 -3563.075} C_VEL
LIN {X 0,Y 545.045,Z 125.589,A -85,B 0,C 180,E1 -3566.327,E2 -3566.327} C_VEL
LIN {X 0,Y 545.034,Z 125.597,A -85,B 0,C 180,E1 -3568.95,E2 -3568.95} C_VEL
LIN {X 0,Y 545.032,Z 125.589,A -85,B 0,C 180,E1 -3571.504,E2 -3571.504} C_VEL
LIN {X 0,Y 545.03,Z 125.596,A -85,B 0,C 180,E1 -3574.506,E2 -3574.506} C_VEL
LIN {X 0,Y 544.987,Z 125.594,A -85,B 0,C 180,E1 -3577.24,E2 -3577.24} C_VEL
LIN {X 0,Y 545.003,Z 125.593,A -85,B 0,C 180,E1 -3579.624,E2 -3579.624} C_VEL
LIN {X 0,Y 545.03,Z 125.593,A -85,B 0,C 180,E1 -3582.748,E2 -3582.748} C_VEL
LIN {X 0,Y 545.044,Z 125.588,A -85,B 0,C 180,E1 -3585.819,E2 -3585.819} C_VEL
LIN {X 0,Y 545.071,Z 125.583,A -85,B 0,C 180,E1 -3588.849,E2 -3588.849} C_VEL
LIN {X 0,Y 545.062,Z 125.59,A -85,B 0,C 180,E1 -3591.846,E2 -3591.846} C_VEL
LIN {X 0,Y 545.158,Z 125.573,A -85,B 0,C 180,E1 -3594.823,E2 -3594.823} C_VEL
LIN {X 0,Y 545.19,Z 125.575,A -85,B 0,C 180,E1 -3597.784,E2 -3597.784} C_VEL
LIN {X 0,Y 545.191,Z 125.576,A -85,B 0,C 180,E1 -3600,E2 -3600} C_VEL
LIN {X 0,Y 545.143,Z 125.572,A -85,B 0,C 180,E1 -3602.956,E2 -3602.956} C_VEL
LIN {X 0,Y 545.127,Z 125.582,A -85,B 0,C 180,E1 -3605.92,E2 -3605.92} C_VEL
LIN {X 0,Y 545.07,Z 125.583,A -85,B 0,C 180,E1 -3608.901,E2 -3608.901} C_VEL
LIN {X 0,Y 545.095,Z 125.582,A -85,B 0,C 180,E1 -3611.905,E2 -3611.905} C_VEL
LIN {X 0,Y 545.078,Z 125.585,A -85,B 0,C 180,E1 -3614.944,E2 -3614.944} C_VEL
LIN {X 0,Y 545.055,Z 125.585,A -85,B 0,C 180,E1 -3618.027,E2 -3618.027} C_VEL
LIN {X 0,Y 545.091,Z 125.581,A -85,B 0,C 180,E1 -3620.372,E2 -3620.372} C_VEL
LIN {X 0,Y 545.072,Z 125.587,A -85,B 0,C 180,E1 -3623.56,E2 -3623.56} C_VEL
LIN {X 0,Y 545.067,Z 125.583,A -85,B 0,C 180,E1 -3626.001,E2 -3626.001} C_VEL
LIN {X 0,Y 545.048,Z 125.592,A -85,B 0,C 180,E1 -3628.74,E2 -3628.74} C_VEL
LIN {X 0,Y 545.059,Z 125.586,A -85,B 0,C 180,E1 -3631.679,E2 -3631.679} C_VEL
LIN {X 0,Y 545.06,Z 125.59,A -85,B 0,C 180,E1 -3634.565,E2 -3634.565} C_VEL
LIN {X 0,Y 545.036,Z 125.589,A -85,B 0,C 180,E1 -3637.304,E2 -3637.304} C_VEL
LIN {X 0,Y 545.066,Z 125.587,A -85,B 0,C 180,E1 -3640.143,E2 -3640.143} C_VEL
LIN {X 0,Y 545.04,Z 125.595,A -85,B 0,C 180,E1 -3642.694,E2 -3642.694} C_VEL
LIN {X 0,Y 545.032,Z 125.59,A -85,B 0,C 180,E1 -3645.171,E2 -3645.171} C_VEL
LIN {X 0,Y 545.064,Z 125.588,A -85,B 0,C 180,E1 -3647.895,E2 -3647.895} C_VEL
LIN {X 0,Y 545.085,Z 125.585,A -85,B 0,C 180,E1 -3650.818,E2 -3650.818} C_VEL
LIN {X 0,Y 545.037,Z 125.59,A -85,B 0,C 180,E1 -3653.619,E2 -3653.619} C_VEL
LIN {X 0,Y 545.068,Z 125.592,A -85,B 0,C 180,E1 -3656.328,E2 -3656.328} C_VEL
LIN {X 0,Y 545.067,Z 125.586,A -85,B 0,C 180,E1 -3658.952,E2 -3658.952} C_VEL
LIN {X 0,Y 545.084,Z 125.586,A -85,B 0,C 180,E1 -3661.506,E2 -3661.506} C_VEL
LIN {X 0,Y 545.097,Z 125.586,A -85,B 0,C 180,E1 -3664.491,E2 -3664.491} C_VEL
LIN {X 0,Y 545.1,Z 125.646,A -85,B 0,C 180,E1 -3665.608,E2 -3665.608} C_VEL
LIN {X 0,Y 546.194,Z 132.698,A -85,B 0,C 180,E1 -3666.692,E2 -3666.692} C_VEL
LIN {X 0,Y 545.997,Z 147.677,A -85,B 0,C 180,E1 -3668.874,E2 -3668.874} C_VEL
LIN {X 0,Y 545.649,Z 169.404,A -85,B 0,C 180,E1 -3671.994,E2 -3671.994} C_VEL
LIN {X 0,Y 545.342,Z 189.7,A -85,B 0,C 180,E1 -3674.872,E2 -3674.872} C_VEL
LIN {X 0,Y 545.307,Z 193.686,A -85,B 0,C 180,E1 -3675.435,E2 -3675.435} C_VEL
LIN {X 0,Y 546.523,Z 203.019,A -85,B 0,C 180,E1 -3675.595,E2 -3675.595} C_VEL
LIN {X 0,Y 546.185,Z 302.139,A -85,B 0,C 180,E1 -3676.915,E2 -3676.915} C_VEL
LIN {X 0,Y 546.024,Z 315.487,A -85,B 0,C 180,E1 -3677.243,E2 -3677.243} C_VEL
LIN {X 0,Y 545.871,Z 327.704,A -85,B 0,C 180,E1 -3677.688,E2 -3677.688} C_VEL
LIN {X 0,Y 545.673,Z 339.131,A -85,B 0,C 180,E1 -3678.245,E2 -3678.245} C_VEL
LIN {X 0,Y 545.497,Z 350.374,A -85,B 0,C 180,E1 -3678.951,E2 -3678.951} C_VEL
LIN {X 0,Y 545.248,Z 361.078,A -85,B 0,C 180,E1 -3679.791,E2 -3679.791} C_VEL
LIN {X 0,Y 545.088,Z 370.728,A -85,B 0,C 180,E1 -3680.725,E2 -3680.725} C_VEL
LIN {X 0,Y 544.947,Z 378.64,A -85,B 0,C 180,E1 -3681.658,E2 -3681.658} C_VEL
LIN {X 0,Y 544.824,Z 386.368,A -85,B 0,C 180,E1 -3682.775,E2 -3682.775} C_VEL
LIN {X 0,Y 544.777,Z 393.493,A -85,B 0,C 180,E1 -3684.076,E2 -3684.076} C_VEL
LIN {X 0,Y 544.629,Z 398.229,A -85,B 0,C 180,E1 -3685.188,E2 -3685.188} C_VEL
LIN {X 0,Y 544.669,Z 401.853,A -85,B 0,C 180,E1 -3686.301,E2 -3686.301} C_VEL
LIN {X 0,Y 544.65,Z 403.721,A -85,B 0,C 180,E1 -3687.041,E2 -3687.041} C_VEL
LIN {X 0,Y 544.546,Z 406.117,A -85,B 0,C 180,E1 -3688.521,E2 -3688.521} C_VEL
LIN {X 0,Y 544.542,Z 406.727,A -85,B 0,C 180,E1 -3689.26,E2 -3689.26} C_VEL
LIN {X 0,Y 544.541,Z 406.944,A -85,B 0,C 180,E1 -3690,E2 -3690} C_VEL
LIN {X 0,Y 544.542,Z 406.728,A -85,B 0,C 180,E1 -3690.739,E2 -3690.739} C_VEL
LIN {X 0,Y 544.572,Z 405.122,A -85,B 0,C 180,E1 -3692.219,E2 -3692.219} C_VEL
LIN {X 0,Y 544.65,Z 403.726,A -85,B 0,C 180,E1 -3692.958,E2 -3692.958} C_VEL
LIN {X 0,Y 544.684,Z 400.783,A -85,B 0,C 180,E1 -3694.069,E2 -3694.069} C_VEL
LIN {X 0,Y 544.653,Z 396.795,A -85,B 0,C 180,E1 -3695.182,E2 -3695.182} C_VEL
LIN {X 0,Y 544.71,Z 391.502,A -85,B 0,C 180,E1 -3696.328,E2 -3696.328} C_VEL
LIN {X 0,Y 544.836,Z 385.211,A -85,B 0,C 180,E1 -3697.411,E2 -3697.411} C_VEL
LIN {X 0,Y 544.972,Z 377.158,A -85,B 0,C 180,E1 -3698.529,E2 -3698.529} C_VEL
LIN {X 0,Y 545.114,Z 368.952,A -85,B 0,C 180,E1 -3699.461,E2 -3699.461} C_VEL
LIN {X 0,Y 545.349,Z 358.951,A -85,B 0,C 180,E1 -3700.394,E2 -3700.394} C_VEL
LIN {X 0,Y 545.53,Z 348.077,A -85,B 0,C 180,E1 -3701.208,E2 -3701.208} C_VEL
LIN {X 0,Y 545.709,Z 336.593,A -85,B 0,C 180,E1 -3701.891,E2 -3701.891} C_VEL
LIN {X 0,Y 545.922,Z 324.337,A -85,B 0,C 180,E1 -3702.453,E2 -3702.453} C_VEL
LIN {X 0,Y 546.104,Z 311.467,A -85,B 0,C 180,E1 -3702.873,E2 -3702.873} C_VEL
LIN {X 0,Y 546.212,Z 297.81,A -85,B 0,C 180,E1 -3703.155,E2 -3703.155} C_VEL
LIN {X 0,Y 546.344,Z 200.83,A -85,B 0,C 180,E1 -3704.44,E2 -3704.44} C_VEL
LIN {X 0,Y 545.324,Z 193.66,A -85,B 0,C 180,E1 -3704.58,E2 -3704.58} C_VEL
LIN {X 0,Y 545.593,Z 173.287,A -85,B 0,C 180,E1 -3707.475,E2 -3707.475} C_VEL
LIN {X 0,Y 545.927,Z 153.324,A -85,B 0,C 180,E1 -3710.34,E2 -3710.34} C_VEL
LIN {X 0,Y 546.281,Z 134.383,A -85,B 0,C 180,E1 -3713.103,E2 -3713.103} C_VEL
LIN {X 0,Y 545.797,Z 129.134,A -85,B 0,C 180,E1 -3713.902,E2 -3713.902} C_VEL
LIN {X 0,Y 545.108,Z 125.587,A -85,B 0,C 180,E1 -3714.468,E2 -3714.468} C_VEL
LIN {X 0,Y 545.082,Z 125.584,A -85,B 0,C 180,E1 -3717.17,E2 -3717.17} C_VEL
LIN {X 0,Y 545.08,Z 125.59,A -85,B 0,C 180,E1 -3720.246,E2 -3720.246} C_VEL
LIN {X 0,Y 545.081,Z 125.582,A -85,B 0,C 180,E1 -3723.062,E2 -3723.062} C_VEL
LIN {X 0,Y 545.035,Z 125.593,A -85,B 0,C 180,E1 -3725.673,E2 -3725.673} C_VEL
LIN {X 0,Y 545.054,Z 125.589,A -85,B 0,C 180,E1 -3728.237,E2 -3728.237} C_VEL
LIN {X 0,Y 545.083,Z 125.583,A -85,B 0,C 180,E1 -3730.473,E2 -3730.473} C_VEL
LIN {X 0,Y 545.079,Z 125.583,A -85,B 0,C 180,E1 -3733.106,E2 -3733.106} C_VEL
LIN {X 0,Y 545.068,Z 125.586,A -85,B 0,C 180,E1 -3736.224,E2 -3736.224} C_VEL
LIN {X 0,Y 545.082,Z 125.582,A -85,B 0,C 180,E1 -3738.885,E2 -3738.885} C_VEL
LIN {X 0,Y 545.081,Z 125.583,A -85,B 0,C 180,E1 -3740.818,E2 -3740.818} C_VEL
LIN {X 0,Y 545.043,Z 125.595,A -85,B 0,C 180,E1 -3743.619,E2 -3743.619} C_VEL
LIN {X 0,Y 545.051,Z 125.586,A -85,B 0,C 180,E1 -3746.327,E2 -3746.327} C_VEL
LIN {X 0,Y 545.065,Z 125.587,A -85,B 0,C 180,E1 -3748.952,E2 -3748.952} C_VEL
LIN {X 0,Y 545.102,Z 125.586,A -85,B 0,C 180,E1 -3751.507,E2 -3751.507} C_VEL
LIN {X 0,Y 545.095,Z 125.581,A -85,B 0,C 180,E1 -3754.491,E2 -3754.491} C_VEL
LIN {X 0,Y 545.038,Z 125.596,A -85,B 0,C 180,E1 -3757.242,E2 -3757.242} C_VEL
LIN {X 0,Y 545.117,Z 125.578,A -85,B 0,C 180,E1 -3760.415,E2 -3760.415} C_VEL
LIN {X 0,Y 545.069,Z 125.586,A -85,B 0,C 180,E1 -3763.521,E2 -3763.521} C_VEL
LIN {X 0,Y 545.095,Z 125.581,A -85,B 0,C 180,E1 -3765.82,E2 -3765.82} C_VEL
LIN {X 0,Y 545.118,Z 125.585,A -85,B 0,C 180,E1 -3768.849,E2 -3768.849} C_VEL
LIN {X 0,Y 545.098,Z 125.58,A -85,B 0,C 180,E1 -3771.846,E2 -3771.846} C_VEL
LIN {X 0,Y 545.202,Z 125.576,A -85,B 0,C 180,E1 -3774.823,E2 -3774.823} C_VEL
LIN {X 0,Y 545.197,Z 125.568,A -85,B 0,C 180,E1 -3777.784,E2 -3777.784} C_VEL
LIN {X 0,Y 545.213,Z 125.574,A -85,B 0,C 180,E1 -3780.738,E2 -3780.738} C_VEL
LIN {X 0,Y 545.17,Z 125.575,A -85,B 0,C 180,E1 -3782.956,E2 -3782.956} C_VEL
LIN {X 0,Y 545.17,Z 125.572,A -85,B 0,C 180,E1 -3785.919,E2 -3785.919} C_VEL
LIN {X 0,Y 545.11,Z 125.582,A -85,B 0,C 180,E1 -3788.9,E2 -3788.9} C_VEL
LIN {X 0,Y 545.134,Z 125.578,A -85,B 0,C 180,E1 -3791.904,E2 -3791.904} C_VEL
LIN {X 0,Y 545.085,Z 125.583,A -85,B 0,C 180,E1 -3794.943,E2 -3794.943} C_VEL
LIN {X 0,Y 545.07,Z 125.589,A -85,B 0,C 180,E1 -3798.026,E2 -3798.026} C_VEL
LIN {X 0,Y 545.092,Z 125.588,A -85,B 0,C 180,E1 -3800.372,E2 -3800.372} C_VEL
LIN {X 0,Y 545.079,Z 125.584,A -85,B 0,C 180,E1 -3803.559,E2 -3803.559} C_VEL
LIN {X 0,Y 545.077,Z 125.59,A -85,B 0,C 180,E1 -3806.001,E2 -3806.001} C_VEL
LIN {X 0,Y 545.073,Z 125.584,A -85,B 0,C 180,E1 -3808.745,E2 -3808.745} C_VEL
LIN {X 0,Y 545.057,Z 125.59,A -85,B 0,C 180,E1 -3811.679,E2 -3811.679} C_VEL
LIN {X 0,Y 545.061,Z 125.586,A -85,B 0,C 180,E1 -3814.564,E2 -3814.564} C_VEL
LIN {X 0,Y 545.06,Z 125.585,A -85,B 0,C 180,E1 -3817.008,E2 -3817.008} C_VEL
LIN {X 0,Y 544.354,Z 125.68,A -85,B 0,C 180,E1 -3817.624,E2 -3817.624} C_VEL
LIN {X 0,Y 541.491,Z 126.037,A -85,B 0,C 180,E1 -3818.625,E2 -3818.625} C_VEL
LIN {X 0,Y 539.104,Z 126.334,A -85,B 0,C 180,E1 -3819.431,E2 -3819.431} C_VEL
LIN {X 0,Y 538.094,Z 126.458,A -85,B 0,C 180,E1 -3820.053,E2 -3820.053} C_VEL
LIN {X 0,Y 538.018,Z 126.464,A -85,B 0,C 180,E1 -3820.264,E2 -3820.264} C_VEL
LIN {X 0,Y 538.025,Z 126.462,A -85,B 0,C 180,E1 -3822.987,E2 -3822.987} C_VEL
LIN {X 0,Y 538.019,Z 126.464,A -85,B 0,C 180,E1 -3826.186,E2 -3826.186} C_VEL
LIN {X 0,Y 538.047,Z 126.463,A -85,B 0,C 180,E1 -3829.253,E2 -3829.253} C_VEL
LIN {X 0,Y 537.991,Z 126.467,A -85,B 0,C 180,E1 -3832.122,E2 -3832.122} C_VEL
LIN {X 0,Y 537.996,Z 126.467,A -85,B 0,C 180,E1 -3834.916,E2 -3834.916} C_VEL
LIN {X 0,Y 538.016,Z 126.468,A -85,B 0,C 180,E1 -3837.617,E2 -3837.617} C_VEL
LIN {X 0,Y 538.014,Z 126.462,A -85,B 0,C 180,E1 -3840.239,E2 -3840.239} C_VEL
LIN {X 0,Y 538.054,Z 126.46,A -85,B 0,C 180,E1 -3842.796,E2 -3842.796} C_VEL
LIN {X 0,Y 538.046,Z 126.466,A -85,B 0,C 180,E1 -3845.293,E2 -3845.293} C_VEL
LIN {X 0,Y 538.022,Z 126.463,A -85,B 0,C 180,E1 -3848.546,E2 -3848.546} C_VEL
LIN {X 0,Y 538.031,Z 126.468,A -85,B 0,C 180,E1 -3850.94,E2 -3850.94} C_VEL
LIN {X 0,Y 538.016,Z 126.467,A -85,B 0,C 180,E1 -3853.299,E2 -3853.299} C_VEL
LIN {X 0,Y 538.06,Z 126.458,A -85,B 0,C 180,E1 -3855.631,E2 -3855.631} C_VEL
LIN {X 0,Y 538.077,Z 126.461,A -85,B 0,C 180,E1 -3858.702,E2 -3858.702} C_VEL
LIN {X 0,Y 538.062,Z 126.456,A -85,B 0,C 180,E1 -3861.739,E2 -3861.739} C_VEL
LIN {X 0,Y 538.16,Z 126.454,A -85,B 0,C 180,E1 -3864.755,E2 -3864.755} C_VEL
LIN {X 0,Y 538.168,Z 126.445,A -85,B 0,C 180,E1 -3867.755,E2 -3867.755} C_VEL
LIN {X 0,Y 538.181,Z 126.451,A -85,B 0,C 180,E1 -3870.748,E2 -3870.748} C_VEL
LIN {X 0,Y 538.101,Z 126.668,A -85,B 0,C 180,E1 -3871.263,E2 -3871.263} C_VEL
LIN {X 0,Y 538.45,Z 131.704,A -85,B 0,C 180,E1 -3872.244,E2 -3872.244} C_VEL
LIN {X 0,Y 538.237,Z 147.891,A -85,B 0,C 180,E1 -3875.315,E2 -3875.315} C_VEL
LIN {X 0,Y 539.635,Z 156.011,A -85,B 0,C 180,E1 -3875.465,E2 -3875.465} C_VEL
LIN {X 0,Y 539.273,Z 254.436,A -85,B 0,C 180,E1 -3876.802,E2 -3876.802} C_VEL
LIN {X 0,Y 539.135,Z 267.633,A -85,B 0,C 180,E1 -3877.137,E2 -3877.137} C_VEL
LIN {X 0,Y 538.975,Z 280.236,A -85,B 0,C 180,E1 -3877.612,E2 -3877.612} C_VEL
LIN {X 0,Y 538.794,Z 292.553,A -85,B 0,C 180,E1 -3878.25,E2 -3878.25} C_VEL
LIN {X 0,Y 538.526,Z 303.959,A -85,B 0,C 180,E1 -3879.01,E2 -3879.01} C_VEL
LIN {X 0,Y 538.293,Z 314.239,A -85,B 0,C 180,E1 -3879.867,E2 -3879.867} C_VEL
LIN {X 0,Y 538.064,Z 324.292,A -85,B 0,C 180,E1 -3880.918,E2 -3880.918} C_VEL
LIN {X 0,Y 537.916,Z 331.935,A -85,B 0,C 180,E1 -3881.897,E2 -3881.897} C_VEL
LIN {X 0,Y 537.755,Z 339.156,A -85,B 0,C 180,E1 -3883.029,E2 -3883.029} C_VEL
LIN {X 0,Y 537.692,Z 344.135,A -85,B 0,C 180,E1 -3883.993,E2 -3883.993} C_VEL
LIN {X 0,Y 537.626,Z 348.974,A -85,B 0,C 180,E1 -3885.156,E2 -3885.156} C_VEL
LIN {X 0,Y 537.549,Z 352.672,A -85,B 0,C 180,E1 -3886.326,E2 -3886.326} C_VEL
LIN {X 0,Y 537.49,Z 355.305,A -85,B 0,C 180,E1 -3887.502,E2 -3887.502} C_VEL
LIN {X 0,Y 537.473,Z 356.51,A -85,B 0,C 180,E1 -3888.29,E2 -3888.29} C_VEL
LIN {X 0,Y 537.491,Z 357.525,A -85,B 0,C 180,E1 -3889.705,E2 -3889.705} C_VEL
LIN {X 0,Y 537.493,Z 357.454,A -85,B 0,C 180,E1 -3890.673,E2 -3890.673} C_VEL
LIN {X 0,Y 537.485,Z 356.493,A -85,B 0,C 180,E1 -3891.817,E2 -3891.817} C_VEL
LIN {X 0,Y 537.515,Z 354.317,A -85,B 0,C 180,E1 -3893.095,E2 -3893.095} C_VEL
LIN {X 0,Y 537.593,Z 351.076,A -85,B 0,C 180,E1 -3894.318,E2 -3894.318} C_VEL
LIN {X 0,Y 537.65,Z 346.433,A -85,B 0,C 180,E1 -3895.585,E2 -3895.585} C_VEL
LIN {X 0,Y 537.755,Z 340.608,A -85,B 0,C 180,E1 -3896.801,E2 -3896.801} C_VEL
LIN {X 0,Y 537.89,Z 334.328,A -85,B 0,C 180,E1 -3897.848,E2 -3897.848} C_VEL
LIN {X 0,Y 538.039,Z 326.347,A -85,B 0,C 180,E1 -3898.935,E2 -3898.935} C_VEL
LIN {X 0,Y 538.246,Z 316.952,A -85,B 0,C 180,E1 -3899.963,E2 -3899.963} C_VEL
LIN {X 0,Y 538.476,Z 306.052,A -85,B 0,C 180,E1 -3900.925,E2 -3900.925} C_VEL
LIN {X 0,Y 538.695,Z 295.978,A -85,B 0,C 180,E1 -3901.637,E2 -3901.637} C_VEL
LIN {X 0,Y 538.949,Z 283.629,A -85,B 0,C 180,E1 -3902.32,E2 -3902.32} C_VEL
LIN {X 0,Y 539.121,Z 270.502,A -85,B 0,C 180,E1 -3902.863,E2 -3902.863} C_VEL
LIN {X 0,Y 539.311,Z 257.354,A -85,B 0,C 180,E1 -3903.226,E2 -3903.226} C_VEL
LIN {X 0,Y 539.393,Z 239.976,A -85,B 0,C 180,E1 -3903.5,E2 -3903.5} C_VEL
LIN {X 0,Y 539.569,Z 154.967,A -85,B 0,C 180,E1 -3904.642,E2 -3904.642} C_VEL
LIN {X 0,Y 538.213,Z 147.688,A -85,B 0,C 180,E1 -3904.786,E2 -3904.786} C_VEL
LIN {X 0,Y 538.395,Z 133.442,A -85,B 0,C 180,E1 -3907.493,E2 -3907.493} C_VEL
LIN {X 0,Y 538.103,Z 126.733,A -85,B 0,C 180,E1 -3908.774,E2 -3908.774} C_VEL
LIN {X 0,Y 538.048,Z 126.466,A -85,B 0,C 180,E1 -3908.828,E2 -3908.828} C_VEL
LIN {X 0,Y 537.989,Z 126.47,A -85,B 0,C 180,E1 -3911.874,E2 -3911.874} C_VEL
LIN {X 0,Y 537.993,Z 126.471,A -85,B 0,C 180,E1 -3914.864,E2 -3914.864} C_VEL
LIN {X 0,Y 537.974,Z 126.476,A -85,B 0,C 180,E1 -3917.21,E2 -3917.21} C_VEL
LIN {X 0,Y 538.007,Z 126.463,A -85,B 0,C 180,E1 -3920.202,E2 -3920.202} C_VEL
LIN {X 0,Y 538.018,Z 126.468,A -85,B 0,C 180,E1 -3923.067,E2 -3923.067} C_VEL
LIN {X 0,Y 537.997,Z 126.466,A -85,B 0,C 180,E1 -3925.825,E2 -3925.825} C_VEL
LIN {X 0,Y 537.99,Z 126.471,A -85,B 0,C 180,E1 -3928.498,E2 -3928.498} C_VEL
LIN {X 0,Y 537.984,Z 126.471,A -85,B 0,C 180,E1 -3931.096,E2 -3931.096} C_VEL
LIN {X 0,Y 537.98,Z 126.468,A -85,B 0,C 180,E1 -3933.63,E2 -3933.63} C_VEL
LIN {X 0,Y 537.983,Z 126.47,A -85,B 0,C 180,E1 -3936.128,E2 -3936.128} C_VEL
LIN {X 0,Y 537.988,Z 126.474,A -85,B 0,C 180,E1 -3938.545,E2 -3938.545} C_VEL
LIN {X 0,Y 537.955,Z 126.472,A -85,B 0,C 180,E1 -3940.937,E2 -3940.937} C_VEL
LIN {X 0,Y 537.966,Z 126.469,A -85,B 0,C 180,E1 -3943.297,E2 -3943.297} C_VEL
LIN {X 0,Y 538.018,Z 126.462,A -85,B 0,C 180,E1 -3945.63,E2 -3945.63} C_VEL
LIN {X 0,Y 538.023,Z 126.462,A -85,B 0,C 180,E1 -3948.701,E2 -3948.701} C_VEL
LIN {X 0,Y 538.031,Z 126.464,A -85,B 0,C 180,E1 -3951.739,E2 -3951.739} C_VEL
LIN {X 0,Y 538.118,Z 126.45,A -85,B 0,C 180,E1 -3954.755,E2 -3954.755} C_VEL
LIN {X 0,Y 538.161,Z 126.45,A -85,B 0,C 180,E1 -3957.755,E2 -3957.755} C_VEL
LIN {X 0,Y 538.16,Z 126.452,A -85,B 0,C 180,E1 -3960,E2 -3960} C_VEL
LIN {X 0,Y 538.111,Z 126.448,A -85,B 0,C 180,E1 -3962.995,E2 -3962.995} C_VEL
LIN {X 0,Y 538.082,Z 126.458,A -85,B 0,C 180,E1 -3965.998,E2 -3965.998} C_VEL
LIN {X 0,Y 538.029,Z 126.461,A -85,B 0,C 180,E1 -3969.018,E2 -3969.018} C_VEL
LIN {X 0,Y 538.054,Z 126.457,A -85,B 0,C 180,E1 -3972.063,E2 -3972.063} C_VEL
LIN {X 0,Y 538.039,Z 126.464,A -85,B 0,C 180,E1 -3975.144,E2 -3975.144} C_VEL
LIN {X 0,Y 538.009,Z 126.461,A -85,B 0,C 180,E1 -3978.271,E2 -3978.271} C_VEL
LIN {X 0,Y 538.037,Z 126.461,A -85,B 0,C 180,E1 -3980.652,E2 -3980.652} C_VEL
LIN {X 0,Y 538.008,Z 126.464,A -85,B 0,C 180,E1 -3983.878,E2 -3983.878} C_VEL
LIN {X 0,Y 538.033,Z 126.46,A -85,B 0,C 180,E1 -3986.367,E2 -3986.367} C_VEL
LIN {X 0,Y 537.994,Z 126.474,A -85,B 0,C 180,E1 -3988.926,E2 -3988.926} C_VEL
LIN {X 0,Y 538.01,Z 126.463,A -85,B 0,C 180,E1 -3991.887,E2 -3991.887} C_VEL
LIN {X 0,Y 538.01,Z 126.469,A -85,B 0,C 180,E1 -3994.617,E2 -3994.617} C_VEL
LIN {X 0,Y 538.005,Z 126.466,A -85,B 0,C 180,E1 -3997.17,E2 -3997.17} C_VEL
LIN {X 0,Y 538.012,Z 126.464,A -85,B 0,C 180,E1 -3999.798,E2 -3999.798} C_VEL
LIN {X 0,Y 537.99,Z 126.472,A -85,B 0,C 180,E1 -4002.789,E2 -4002.789} C_VEL
LIN {X 0,Y 538.003,Z 126.466,A -85,B 0,C 180,E1 -4005.137,E2 -4005.137} C_VEL
LIN {X 0,Y 538.021,Z 126.47,A -85,B 0,C 180,E1 -4008.226,E2 -4008.226} C_VEL
LIN {X 0,Y 538.016,Z 126.464,A -85,B 0,C 180,E1 -4011.17,E2 -4011.17} C_VEL
LIN {X 0,Y 537.992,Z 126.473,A -85,B 0,C 180,E1 -4014.089,E2 -4014.089} C_VEL
LIN {X 0,Y 538.034,Z 126.463,A -85,B 0,C 180,E1 -4016.727,E2 -4016.727} C_VEL
LIN {X 0,Y 538.015,Z 126.467,A -85,B 0,C 180,E1 -4019.559,E2 -4019.559} C_VEL
LIN {X 0,Y 538.047,Z 126.462,A -85,B 0,C 180,E1 -4022.651,E2 -4022.651} C_VEL
LIN {X 0,Y 538.096,Z 126.587,A -85,B 0,C 180,E1 -4025.46,E2 -4025.46} C_VEL
LIN {X 0,Y 539.256,Z 133.726,A -85,B 0,C 180,E1 -4026.578,E2 -4026.578} C_VEL
LIN {X 0,Y 538.987,Z 151.409,A -85,B 0,C 180,E1 -4029.187,E2 -4029.187} C_VEL
LIN {X 0,Y 538.582,Z 172.759,A -85,B 0,C 180,E1 -4032.286,E2 -4032.286} C_VEL
LIN {X 0,Y 538.297,Z 192.001,A -85,B 0,C 180,E1 -4035.049,E2 -4035.049} C_VEL
LIN {X 0,Y 538.265,Z 193.299,A -85,B 0,C 180,E1 -4035.234,E2 -4035.234} C_VEL
LIN {X 0,Y 539.639,Z 204.357,A -85,B 0,C 180,E1 -4035.429,E2 -4035.429} C_VEL
LIN {X 0,Y 539.276,Z 301.738,A -85,B 0,C 180,E1 -4036.745,E2 -4036.745} C_VEL
LIN {X 0,Y 539.098,Z 315.109,A -85,B 0,C 180,E1 -4037.076,E2 -4037.076} C_VEL
LIN {X 0,Y 538.889,Z 328.465,A -85,B 0,C 180,E1 -4037.573,E2 -4037.573} C_VEL
LIN {X 0,Y 538.681,Z 339.331,A -85,B 0,C 180,E1 -4038.122,E2 -4038.122} C_VEL
LIN {X 0,Y 538.434,Z 351.318,A -85,B 0,C 180,E1 -4038.9,E2 -4038.9} C_VEL
LIN {X 0,Y 538.192,Z 361.805,A -85,B 0,C 180,E1 -4039.751,E2 -4039.751} C_VEL
LIN {X 0,Y 538.048,Z 370.383,A -85,B 0,C 180,E1 -4040.603,E2 -4040.603} C_VEL
LIN {X 0,Y 537.892,Z 378.299,A -85,B 0,C 180,E1 -4041.547,E2 -4041.547} C_VEL
LIN {X 0,Y 537.755,Z 386.03,A -85,B 0,C 180,E1 -4042.679,E2 -4042.679} C_VEL
LIN {X 0,Y 537.665,Z 393.158,A -85,B 0,C 180,E1 -4043.997,E2 -4043.997} C_VEL
LIN {X 0,Y 537.54,Z 397.897,A -85,B 0,C 180,E1 -4045.125,E2 -4045.125} C_VEL
LIN {X 0,Y 537.591,Z 401.525,A -85,B 0,C 180,E1 -4046.252,E2 -4046.252} C_VEL
LIN {X 0,Y 537.58,Z 403.395,A -85,B 0,C 180,E1 -4047.002,E2 -4047.002} C_VEL
LIN {X 0,Y 537.452,Z 405.792,A -85,B 0,C 180,E1 -4048.501,E2 -4048.501} C_VEL
LIN {X 0,Y 537.449,Z 406.402,A -85,B 0,C 180,E1 -4049.251,E2 -4049.251} C_VEL
LIN {X 0,Y 537.449,Z 406.621,A -85,B 0,C 180,E1 -4050,E2 -4050} C_VEL
LIN {X 0,Y 537.449,Z 406.405,A -85,B 0,C 180,E1 -4050.749,E2 -4050.749} C_VEL
LIN {X 0,Y 537.49,Z 404.8,A -85,B 0,C 180,E1 -4052.248,E2 -4052.248} C_VEL
LIN {X 0,Y 537.58,Z 403.404,A -85,B 0,C 180,E1 -4052.997,E2 -4052.997} C_VEL
LIN {X 0,Y 537.603,Z 400.46,A -85,B 0,C 180,E1 -4054.123,E2 -4054.123} C_VEL
LIN {X 0,Y 537.587,Z 396.472,A -85,B 0,C 180,E1 -4055.25,E2 -4055.25} C_VEL
LIN {X 0,Y 537.645,Z 390.409,A -85,B 0,C 180,E1 -4056.555,E2 -4056.555} C_VEL
LIN {X 0,Y 537.784,Z 383.643,A -85,B 0,C 180,E1 -4057.698,E2 -4057.698} C_VEL
LIN {X 0,Y 537.931,Z 375.332,A -85,B 0,C 180,E1 -4058.83,E2 -4058.83} C_VEL
LIN {X 0,Y 538.091,Z 366.814,A -85,B 0,C 180,E1 -4059.776,E2 -4059.776} C_VEL
LIN {X 0,Y 538.351,Z 356.293,A -85,B 0,C 180,E1 -4060.721,E2 -4060.721} C_VEL
LIN {X 0,Y 538.582,Z 345.086,A -85,B 0,C 180,E1 -4061.531,E2 -4061.531} C_VEL
LIN {X 0,Y 538.809,Z 334.479,A -85,B 0,C 180,E1 -4062.141,E2 -4062.141} C_VEL
LIN {X 0,Y 538.984,Z 322.763,A -85,B 0,C 180,E1 -4062.663,E2 -4062.663} C_VEL
LIN {X 0,Y 539.208,Z 310.186,A -85,B 0,C 180,E1 -4063.065,E2 -4063.065} C_VEL
LIN {X 0,Y 539.316,Z 297.418,A -85,B 0,C 180,E1 -4063.326,E2 -4063.326} C_VEL
LIN {X 0,Y 539.511,Z 201.802,A -85,B 0,C 180,E1 -4064.61,E2 -4064.61} C_VEL
LIN {X 0,Y 538.29,Z 193.397,A -85,B 0,C 180,E1 -4064.766,E2 -4064.766} C_VEL
LIN {X 0,Y 538.583,Z 174.673,A -85,B 0,C 180,E1 -4067.465,E2 -4067.465} C_VEL
LIN {X 0,Y 538.953,Z 154.084,A -85,B 0,C 180,E1 -4070.458,E2 -4070.458} C_VEL
LIN {X 0,Y 539.36,Z 135.451,A -85,B 0,C 180,E1 -4073.214,E2 -4073.214} C_VEL
LIN {X 0,Y 538.75,Z 130.024,A -85,B 0,C 180,E1 -4074.055,E2 -4074.055} C_VEL
LIN {X 0,Y 538.053,Z 126.465,A -85,B 0,C 180,E1 -4074.661,E2 -4074.661} C_VEL
LIN {X 0,Y 538.046,Z 126.461,A -85,B 0,C 180,E1 -4077.349,E2 -4077.349} C_VEL
LIN {X 0,Y 538.028,Z 126.466,A -85,B 0,C 180,E1 -4080.444,E2 -4080.444} C_VEL
LIN {X 0,Y 538.047,Z 126.459,A -85,B 0,C 180,E1 -4083.283,E2 -4083.283} C_VEL
LIN {X 0,Y 537.996,Z 126.473,A -85,B 0,C 180,E1 -4086.004,E2 -4086.004} C_VEL
LIN {X 0,Y 538.016,Z 126.462,A -85,B 0,C 180,E1 -4088.83,E2 -4088.83} C_VEL
LIN {X 0,Y 538.031,Z 126.47,A -85,B 0,C 180,E1 -4091.773,E2 -4091.773} C_VEL
LIN {X 0,Y 538.008,Z 126.463,A -85,B 0,C 180,E1 -4094.862,E2 -4094.862} C_VEL
LIN {X 0,Y 538.019,Z 126.465,A -85,B 0,C 180,E1 -4097.214,E2 -4097.214} C_VEL
LIN {X 0,Y 538.023,Z 126.463,A -85,B 0,C 180,E1 -4100.203,E2 -4100.203} C_VEL
LIN {X 0,Y 538.025,Z 126.464,A -85,B 0,C 180,E1 -4103.067,E2 -4103.067} C_VEL
LIN {X 0,Y 538.011,Z 126.467,A -85,B 0,C 180,E1 -4105.826,E2 -4105.826} C_VEL
LIN {X 0,Y 538.009,Z 126.463,A -85,B 0,C 180,E1 -4108.498,E2 -4108.498} C_VEL
LIN {X 0,Y 538.043,Z 126.464,A -85,B 0,C 180,E1 -4111.099,E2 -4111.099} C_VEL
LIN {X 0,Y 538.042,Z 126.463,A -85,B 0,C 180,E1 -4113.633,E2 -4113.633} C_VEL
LIN {X 0,Y 538.008,Z 126.463,A -85,B 0,C 180,E1 -4116.122,E2 -4116.122} C_VEL
LIN {X 0,Y 538.038,Z 126.466,A -85,B 0,C 180,E1 -4119.348,E2 -4119.348} C_VEL
LIN {X 0,Y 538.036,Z 126.461,A -85,B 0,C 180,E1 -4122.468,E2 -4122.468} C_VEL
LIN {X 0,Y 538.064,Z 126.457,A -85,B 0,C 180,E1 -4125.631,E2 -4125.631} C_VEL
LIN {X 0,Y 538.077,Z 126.46,A -85,B 0,C 180,E1 -4128.701,E2 -4128.701} C_VEL
LIN {X 0,Y 538.062,Z 126.457,A -85,B 0,C 180,E1 -4131.739,E2 -4131.739} C_VEL
LIN {X 0,Y 538.16,Z 126.453,A -85,B 0,C 180,E1 -4134.755,E2 -4134.755} C_VEL
LIN {X 0,Y 538.168,Z 126.443,A -85,B 0,C 180,E1 -4137.755,E2 -4137.755} C_VEL
LIN {X 0,Y 538.183,Z 126.45,A -85,B 0,C 180,E1 -4140.748,E2 -4140.748} C_VEL
LIN {X 0,Y 538.136,Z 126.451,A -85,B 0,C 180,E1 -4142.994,E2 -4142.994} C_VEL
LIN {X 0,Y 538.121,Z 126.451,A -85,B 0,C 180,E1 -4145.997,E2 -4145.997} C_VEL
LIN {X 0,Y 538.06,Z 126.459,A -85,B 0,C 180,E1 -4149.018,E2 -4149.018} C_VEL
LIN {X 0,Y 538.082,Z 126.458,A -85,B 0,C 180,E1 -4152.062,E2 -4152.062} C_VEL
LIN {X 0,Y 538.045,Z 126.459,A -85,B 0,C 180,E1 -4155.144,E2 -4155.144} C_VEL
LIN {X 0,Y 538.024,Z 126.471,A -85,B 0,C 180,E1 -4158.27,E2 -4158.27} C_VEL
LIN {X 0,Y 538.037,Z 126.463,A -85,B 0,C 180,E1 -4160.651,E2 -4160.651} C_VEL
LIN {X 0,Y 538.002,Z 126.469,A -85,B 0,C 180,E1 -4163.888,E2 -4163.888} C_VEL
LIN {X 0,Y 538.039,Z 126.464,A -85,B 0,C 180,E1 -4166.367,E2 -4166.367} C_VEL
LIN {X 0,Y 538.029,Z 126.461,A -85,B 0,C 180,E1 -4168.933,E2 -4168.933} C_VEL
LIN {X 0,Y 538.009,Z 126.471,A -85,B 0,C 180,E1 -4171.887,E2 -4171.887} C_VEL
LIN {X 0,Y 538.011,Z 126.464,A -85,B 0,C 180,E1 -4174.618,E2 -4174.618} C_VEL
LIN {X 0,Y 538.003,Z 126.465,A -85,B 0,C 180,E1 -4177.17,E2 -4177.17} C_VEL
LIN {X 0,Y 538.018,Z 126.464,A -85,B 0,C 180,E1 -4180.264,E2 -4180.264} C_VEL
LIN {X 0,Y 537.368,Z 126.543,A -85,B 0,C 180,E1 -4180.889,E2 -4180.889} C_VEL
LIN {X 0,Y 534.521,Z 126.904,A -85,B 0,C 180,E1 -4181.904,E2 -4181.904} C_VEL
LIN {X 0,Y 532.099,Z 127.209,A -85,B 0,C 180,E1 -4182.721,E2 -4182.721} C_VEL
LIN {X 0,Y 531.05,Z 127.337,A -85,B 0,C 180,E1 -4183.352,E2 -4183.352} C_VEL
LIN {X 0,Y 530.96,Z 127.346,A -85,B 0,C 180,E1 -4183.566,E2 -4183.566} C_VEL
LIN {X 0,Y 530.964,Z 127.341,A -85,B 0,C 180,E1 -4186.505,E2 -4186.505} C_VEL
LIN {X 0,Y 530.98,Z 127.348,A -85,B 0,C 180,E1 -4189.567,E2 -4189.567} C_VEL
LIN {X 0,Y 530.967,Z 127.34,A -85,B 0,C 180,E1 -4192.577,E2 -4192.577} C_VEL
LIN {X 0,Y 530.979,Z 127.346,A -85,B 0,C 180,E1 -4195.31,E2 -4195.31} C_VEL
LIN {X 0,Y 530.965,Z 127.341,A -85,B 0,C 180,E1 -4198.032,E2 -4198.032} C_VEL
LIN {X 0,Y 530.987,Z 127.341,A -85,B 0,C 180,E1 -4200.875,E2 -4200.875} C_VEL
LIN {X 0,Y 531,Z 127.346,A -85,B 0,C 180,E1 -4203.256,E2 -4203.256} C_VEL
LIN {X 0,Y 530.983,Z 127.339,A -85,B 0,C 180,E1 -4205.961,E2 -4205.961} C_VEL
LIN {X 0,Y 530.998,Z 127.345,A -85,B 0,C 180,E1 -4209.062,E2 -4209.062} C_VEL
LIN {X 0,Y 530.984,Z 127.341,A -85,B 0,C 180,E1 -4211.479,E2 -4211.479} C_VEL
LIN {X 0,Y 530.993,Z 127.341,A -85,B 0,C 180,E1 -4214.65,E2 -4214.65} C_VEL
LIN {X 0,Y 531.04,Z 127.331,A -85,B 0,C 180,E1 -4217.775,E2 -4217.775} C_VEL
LIN {X 0,Y 531.017,Z 127.343,A -85,B 0,C 180,E1 -4220.862,E2 -4220.862} C_VEL
LIN {X 0,Y 531.075,Z 127.327,A -85,B 0,C 180,E1 -4223.923,E2 -4223.923} C_VEL
LIN {X 0,Y 531.102,Z 127.331,A -85,B 0,C 180,E1 -4226.966,E2 -4226.966} C_VEL
LIN {X 0,Y 531.144,Z 127.323,A -85,B 0,C 180,E1 -4230,E2 -4230} C_VEL
LIN {X 0,Y 531.069,Z 127.455,A -85,B 0,C 180,E1 -4231.138,E2 -4231.138} C_VEL
LIN {X 0,Y 531.451,Z 133.245,A -85,B 0,C 180,E1 -4232.274,E2 -4232.274} C_VEL
LIN {X 0,Y 531.213,Z 147.881,A -85,B 0,C 180,E1 -4235.1,E2 -4235.1} C_VEL
LIN {X 0,Y 532.845,Z 157.957,A -85,B 0,C 180,E1 -4235.298,E2 -4235.298} C_VEL
LIN {X 0,Y 532.364,Z 254.966,A -85,B 0,C 180,E1 -4236.633,E2 -4236.633} C_VEL
LIN {X 0,Y 532.227,Z 268.256,A -85,B 0,C 180,E1 -4236.978,E2 -4236.978} C_VEL
LIN {X 0,Y 532.064,Z 280.118,A -85,B 0,C 180,E1 -4237.431,E2 -4237.431} C_VEL
LIN {X 0,Y 531.868,Z 292.47,A -85,B 0,C 180,E1 -4238.071,E2 -4238.071} C_VEL
LIN {X 0,Y 531.588,Z 303.947,A -85,B 0,C 180,E1 -4238.841,E2 -4238.841} C_VEL
LIN {X 0,Y 531.33,Z 314.293,A -85,B 0,C 180,E1 -4239.709,E2 -4239.709} C_VEL
LIN {X 0,Y 531.092,Z 323.588,A -85,B 0,C 180,E1 -4240.677,E2 -4240.677} C_VEL
LIN {X 0,Y 530.888,Z 332.65,A -85,B 0,C 180,E1 -4241.846,E2 -4241.846} C_VEL
LIN {X 0,Y 530.688,Z 339.905,A -85,B 0,C 180,E1 -4243.011,E2 -4243.011} C_VEL
LIN {X 0,Y 530.626,Z 345.689,A -85,B 0,C 180,E1 -4244.184,E2 -4244.184} C_VEL
LIN {X 0,Y 530.539,Z 350.245,A -85,B 0,C 180,E1 -4245.363,E2 -4245.363} C_VEL
LIN {X 0,Y 530.472,Z 352.652,A -85,B 0,C 180,E1 -4246.154,E2 -4246.154} C_VEL
LIN {X 0,Y 530.409,Z 355.58,A -85,B 0,C 180,E1 -4247.444,E2 -4247.444} C_VEL
LIN {X 0,Y 530.408,Z 357.117,A -85,B 0,C 180,E1 -4248.542,E2 -4248.542} C_VEL
LIN {X 0,Y 530.405,Z 357.873,A -85,B 0,C 180,E1 -4249.819,E2 -4249.819} C_VEL
LIN {X 0,Y 530.386,Z 357.604,A -85,B 0,C 180,E1 -4250.963,E2 -4250.963} C_VEL
LIN {X 0,Y 530.417,Z 356.671,A -85,B 0,C 180,E1 -4251.952,E2 -4251.952} C_VEL
LIN {X 0,Y 530.453,Z 353.979,A -85,B 0,C 180,E1 -4253.42,E2 -4253.42} C_VEL
LIN {X 0,Y 530.531,Z 350.471,A -85,B 0,C 180,E1 -4254.663,E2 -4254.663} C_VEL
LIN {X 0,Y 530.606,Z 345.668,A -85,B 0,C 180,E1 -4255.919,E2 -4255.919} C_VEL
LIN {X 0,Y 530.732,Z 339.685,A -85,B 0,C 180,E1 -4257.122,E2 -4257.122} C_VEL
LIN {X 0,Y 530.872,Z 332.667,A -85,B 0,C 180,E1 -4258.248,E2 -4258.248} C_VEL
LIN {X 0,Y 531.086,Z 324.451,A -85,B 0,C 180,E1 -4259.316,E2 -4259.316} C_VEL
LIN {X 0,Y 531.328,Z 314.707,A -85,B 0,C 180,E1 -4260.347,E2 -4260.347} C_VEL
LIN {X 0,Y 531.501,Z 303.817,A -85,B 0,C 180,E1 -4261.265,E2 -4261.265} C_VEL
LIN {X 0,Y 531.861,Z 292.264,A -85,B 0,C 180,E1 -4262.036,E2 -4262.036} C_VEL
LIN {X 0,Y 532.106,Z 281.087,A -85,B 0,C 180,E1 -4262.619,E2 -4262.619} C_VEL
LIN {X 0,Y 532.251,Z 268.204,A -85,B 0,C 180,E1 -4263.116,E2 -4263.116} C_VEL
LIN {X 0,Y 532.429,Z 254.964,A -85,B 0,C 180,E1 -4263.457,E2 -4263.457} C_VEL
LIN {X 0,Y 532.742,Z 155.784,A -85,B 0,C 180,E1 -4264.827,E2 -4264.827} C_VEL
LIN {X 0,Y 531.239,Z 147.882,A -85,B 0,C 180,E1 -4265.001,E2 -4265.001} C_VEL
LIN {X 0,Y 531.437,Z 132.436,A -85,B 0,C 180,E1 -4267.947,E2 -4267.947} C_VEL
LIN {X 0,Y 531.006,Z 127.344,A -85,B 0,C 180,E1 -4268.958,E2 -4268.958} C_VEL
LIN {X 0,Y 530.924,Z 127.348,A -85,B 0,C 180,E1 -4272.159,E2 -4272.159} C_VEL
LIN {X 0,Y 530.966,Z 127.344,A -85,B 0,C 180,E1 -4274.549,E2 -4274.549} C_VEL
LIN {X 0,Y 530.919,Z 127.353,A -85,B 0,C 180,E1 -4277.538,E2 -4277.538} C_VEL
LIN {X 0,Y 530.968,Z 127.342,A -85,B 0,C 180,E1 -4280.555,E2 -4280.555} C_VEL
LIN {X 0,Y 530.95,Z 127.345,A -85,B 0,C 180,E1 -4283.441,E2 -4283.441} C_VEL
LIN {X 0,Y 530.961,Z 127.345,A -85,B 0,C 180,E1 -4286.501,E2 -4286.501} C_VEL
LIN {X 0,Y 530.943,Z 127.347,A -85,B 0,C 180,E1 -4289.361,E2 -4289.361} C_VEL
LIN {X 0,Y 530.93,Z 127.346,A -85,B 0,C 180,E1 -4291.541,E2 -4291.541} C_VEL
LIN {X 0,Y 530.96,Z 127.344,A -85,B 0,C 180,E1 -4294.168,E2 -4294.168} C_VEL
LIN {X 0,Y 530.922,Z 127.354,A -85,B 0,C 180,E1 -4296.602,E2 -4296.602} C_VEL
LIN {X 0,Y 530.93,Z 127.348,A -85,B 0,C 180,E1 -4299.059,E2 -4299.059} C_VEL
LIN {X 0,Y 530.971,Z 127.347,A -85,B 0,C 180,E1 -4302.364,E2 -4302.364} C_VEL
LIN {X 0,Y 530.973,Z 127.338,A -85,B 0,C 180,E1 -4305.435,E2 -4305.435} C_VEL
LIN {X 0,Y 530.986,Z 127.34,A -85,B 0,C 180,E1 -4308.549,E2 -4308.549} C_VEL
LIN {X 0,Y 530.979,Z 127.341,A -85,B 0,C 180,E1 -4311.628,E2 -4311.628} C_VEL
LIN {X 0,Y 531.08,Z 127.327,A -85,B 0,C 180,E1 -4314.685,E2 -4314.685} C_VEL
LIN {X 0,Y 531.133,Z 127.325,A -85,B 0,C 180,E1 -4317.725,E2 -4317.725} C_VEL
LIN {X 0,Y 531.128,Z 127.327,A -85,B 0,C 180,E1 -4320,E2 -4320} C_VEL
LIN {X 0,Y 531.133,Z 127.319,A -85,B 0,C 180,E1 -4322.275,E2 -4322.275} C_VEL
LIN {X 0,Y 531.084,Z 127.329,A -85,B 0,C 180,E1 -4325.315,E2 -4325.315} C_VEL
LIN {X 0,Y 530.996,Z 127.336,A -85,B 0,C 180,E1 -4328.372,E2 -4328.372} C_VEL
LIN {X 0,Y 531.051,Z 127.335,A -85,B 0,C 180,E1 -4331.67,E2 -4331.67} C_VEL
LIN {X 0,Y 531.022,Z 127.336,A -85,B 0,C 180,E1 -4334.951,E2 -4334.951} C_VEL
LIN {X 0,Y 530.974,Z 127.341,A -85,B 0,C 180,E1 -4337.724,E2 -4337.724} C_VEL
LIN {X 0,Y 531.027,Z 127.333,A -85,B 0,C 180,E1 -4340.127,E2 -4340.127} C_VEL
LIN {X 0,Y 530.942,Z 127.342,A -85,B 0,C 180,E1 -4342.574,E2 -4342.574} C_VEL
LIN {X 0,Y 530.961,Z 127.35,A -85,B 0,C 180,E1 -4345.06,E2 -4345.06} C_VEL
LIN {X 0,Y 530.967,Z 127.342,A -85,B 0,C 180,E1 -4347.598,E2 -4347.598} C_VEL
LIN {X 0,Y 530.963,Z 127.345,A -85,B 0,C 180,E1 -4350.643,E2 -4350.643} C_VEL
LIN {X 0,Y 530.964,Z 127.341,A -85,B 0,C 180,E1 -4353.5,E2 -4353.5} C_VEL
LIN {X 0,Y 530.957,Z 127.349,A -85,B 0,C 180,E1 -4356.559,E2 -4356.559} C_VEL
LIN {X 0,Y 530.972,Z 127.341,A -85,B 0,C 180,E1 -4359.445,E2 -4359.445} C_VEL
LIN {X 0,Y 530.959,Z 127.35,A -85,B 0,C 180,E1 -4362.459,E2 -4362.459} C_VEL
LIN {X 0,Y 530.977,Z 127.34,A -85,B 0,C 180,E1 -4365.622,E2 -4365.622} C_VEL
LIN {X 0,Y 530.989,Z 127.346,A -85,B 0,C 180,E1 -4368.564,E2 -4368.564} C_VEL
LIN {X 0,Y 530.959,Z 127.343,A -85,B 0,C 180,E1 -4371.529,E2 -4371.529} C_VEL
LIN {X 0,Y 530.953,Z 127.348,A -85,B 0,C 180,E1 -4374.38,E2 -4374.38} C_VEL
LIN {X 0,Y 530.97,Z 127.342,A -85,B 0,C 180,E1 -4377.133,E2 -4377.133} C_VEL
LIN {X 0,Y 530.962,Z 127.349,A -85,B 0,C 180,E1 -4379.802,E2 -4379.802} C_VEL
LIN {X 0,Y 531.012,Z 127.34,A -85,B 0,C 180,E1 -4382.468,E2 -4382.468} C_VEL
LIN {X 0,Y 531.039,Z 127.39,A -85,B 0,C 180,E1 -4385.284,E2 -4385.284} C_VEL
LIN {X 0,Y 532.308,Z 134.771,A -85,B 0,C 180,E1 -4386.46,E2 -4386.46} C_VEL
LIN {X 0,Y 532.068,Z 149.712,A -85,B 0,C 180,E1 -4388.7,E2 -4388.7} C_VEL
LIN {X 0,Y 531.642,Z 171.362,A -85,B 0,C 180,E1 -4391.892,E2 -4391.892} C_VEL
LIN {X 0,Y 531.277,Z 191.822,A -85,B 0,C 180,E1 -4394.871,E2 -4394.871} C_VEL
LIN {X 0,Y 531.251,Z 192.978,A -85,B 0,C 180,E1 -4395.038,E2 -4395.038} C_VEL
LIN {X 0,Y 532.753,Z 204.015,A -85,B 0,C 180,E1 -4395.237,E2 -4395.237} C_VEL
LIN {X 0,Y 532.364,Z 301.335,A -85,B 0,C 180,E1 -4396.569,E2 -4396.569} C_VEL
LIN {X 0,Y 532.156,Z 314.73,A -85,B 0,C 180,E1 -4396.904,E2 -4396.904} C_VEL
LIN {X 0,Y 531.952,Z 328.098,A -85,B 0,C 180,E1 -4397.409,E2 -4397.409} C_VEL
LIN {X 0,Y 531.709,Z 339.436,A -85,B 0,C 180,E1 -4397.992,E2 -4397.992} C_VEL
LIN {X 0,Y 531.435,Z 350.965,A -85,B 0,C 180,E1 -4398.751,E2 -4398.751} C_VEL
LIN {X 0,Y 531.196,Z 361.457,A -85,B 0,C 180,E1 -4399.615,E2 -4399.615} C_VEL
LIN {X 0,Y 530.985,Z 370.038,A -85,B 0,C 180,E1 -4400.477,E2 -4400.477} C_VEL
LIN {X 0,Y 530.818,Z 377.957,A -85,B 0,C 180,E1 -4401.434,E2 -4401.434} C_VEL
LIN {X 0,Y 530.666,Z 385.692,A -85,B 0,C 180,E1 -4402.581,E2 -4402.581} C_VEL
LIN {X 0,Y 530.56,Z 392.823,A -85,B 0,C 180,E1 -4403.917,E2 -4403.917} C_VEL
LIN {X 0,Y 530.459,Z 397.566,A -85,B 0,C 180,E1 -4405.06,E2 -4405.06} C_VEL
LIN {X 0,Y 530.516,Z 401.197,A -85,B 0,C 180,E1 -4406.202,E2 -4406.202} C_VEL
LIN {X 0,Y 530.483,Z 403.067,A -85,B 0,C 180,E1 -4406.962,E2 -4406.962} C_VEL
LIN {X 0,Y 530.412,Z 404.467,A -85,B 0,C 180,E1 -4407.722,E2 -4407.722} C_VEL
LIN {X 0,Y 530.356,Z 406.078,A -85,B 0,C 180,E1 -4409.241,E2 -4409.241} C_VEL
LIN {X 0,Y 530.357,Z 406.298,A -85,B 0,C 180,E1 -4410,E2 -4410} C_VEL
LIN {X 0,Y 530.356,Z 406.082,A -85,B 0,C 180,E1 -4410.759,E2 -4410.759} C_VEL
LIN {X 0,Y 530.412,Z 404.478,A -85,B 0,C 180,E1 -4412.278,E2 -4412.278} C_VEL
LIN {X 0,Y 530.483,Z 403.081,A -85,B 0,C 180,E1 -4413.038,E2 -4413.038} C_VEL
LIN {X 0,Y 530.521,Z 400.137,A -85,B 0,C 180,E1 -4414.178,E2 -4414.178} C_VEL
LIN {X 0,Y 530.522,Z 396.149,A -85,B 0,C 180,E1 -4415.321,E2 -4415.321} C_VEL
LIN {X 0,Y 530.544,Z 390.682,A -85,B 0,C 180,E1 -4416.53,E2 -4416.53} C_VEL
LIN {X 0,Y 530.682,Z 384.556,A -85,B 0,C 180,E1 -4417.61,E2 -4417.61} C_VEL
LIN {X 0,Y 530.832,Z 376.499,A -85,B 0,C 180,E1 -4418.757,E2 -4418.757} C_VEL
LIN {X 0,Y 531.026,Z 368.29,A -85,B 0,C 180,E1 -4419.715,E2 -4419.715} C_VEL
LIN {X 0,Y 531.305,Z 358.284,A -85,B 0,C 180,E1 -4420.672,E2 -4420.672} C_VEL
LIN {X 0,Y 531.528,Z 346.838,A -85,B 0,C 180,E1 -4421.545,E2 -4421.545} C_VEL
LIN {X 0,Y 531.789,Z 335.909,A -85,B 0,C 180,E1 -4422.207,E2 -4422.207} C_VEL
LIN {X 0,Y 532.031,Z 323.641,A -85,B 0,C 180,E1 -4422.783,E2 -4422.783} C_VEL
LIN {X 0,Y 532.274,Z 310.736,A -85,B 0,C 180,E1 -4423.214,E2 -4423.214} C_VEL
LIN {X 0,Y 532.425,Z 297.027,A -85,B 0,C 180,E1 -4423.502,E2 -4423.502} C_VEL
LIN {X 0,Y 532.627,Z 202.417,A -85,B 0,C 180,E1 -4424.79,E2 -4424.79} C_VEL
LIN {X 0,Y 531.25,Z 193.057,A -85,B 0,C 180,E1 -4424.97,E2 -4424.97} C_VEL
LIN {X 0,Y 531.616,Z 173.327,A -85,B 0,C 180,E1 -4427.852,E2 -4427.852} C_VEL
LIN {X 0,Y 532.058,Z 151.372,A -85,B 0,C 180,E1 -4431.097,E2 -4431.097} C_VEL
LIN {X 0,Y 532.365,Z 135.137,A -85,B 0,C 180,E1 -4433.537,E2 -4433.537} C_VEL
LIN {X 0,Y 531.042,Z 127.338,A -85,B 0,C 180,E1 -4434.794,E2 -4434.794} C_VEL
LIN {X 0,Y 531.011,Z 127.339,A -85,B 0,C 180,E1 -4437.596,E2 -4437.596} C_VEL
LIN {X 0,Y 530.976,Z 127.342,A -85,B 0,C 180,E1 -4440.645,E2 -4440.645} C_VEL
LIN {X 0,Y 530.989,Z 127.344,A -85,B 0,C 180,E1 -4443.772,E2 -4443.772} C_VEL
LIN {X 0,Y 530.956,Z 127.343,A -85,B 0,C 180,E1 -4446.558,E2 -4446.558} C_VEL
LIN {X 0,Y 530.99,Z 127.341,A -85,B 0,C 180,E1 -4449.443,E2 -4449.443} C_VEL
LIN {X 0,Y 530.979,Z 127.34,A -85,B 0,C 180,E1 -4452.456,E2 -4452.456} C_VEL
LIN {X 0,Y 530.983,Z 127.346,A -85,B 0,C 180,E1 -4455.621,E2 -4455.621} C_VEL
LIN {X 0,Y 530.994,Z 127.337,A -85,B 0,C 180,E1 -4458.564,E2 -4458.564} C_VEL
LIN {X 0,Y 530.958,Z 127.35,A -85,B 0,C 180,E1 -4461.529,E2 -4461.529} C_VEL
LIN {X 0,Y 530.954,Z 127.342,A -85,B 0,C 180,E1 -4464.38,E2 -4464.38} C_VEL
LIN {X 0,Y 530.967,Z 127.345,A -85,B 0,C 180,E1 -4467.133,E2 -4467.133} C_VEL
LIN {X 0,Y 530.962,Z 127.344,A -85,B 0,C 180,E1 -4469.802,E2 -4469.802} C_VEL
LIN {X 0,Y 531.013,Z 127.335,A -85,B 0,C 180,E1 -4472.467,E2 -4472.467} C_VEL
LIN {X 0,Y 531.005,Z 127.34,A -85,B 0,C 180,E1 -4474.942,E2 -4474.942} C_VEL
LIN {X 0,Y 530.972,Z 127.34,A -85,B 0,C 180,E1 -4478.247,E2 -4478.247} C_VEL
LIN {X 0,Y 530.992,Z 127.34,A -85,B 0,C 180,E1 -4480.677,E2 -4480.677} C_VEL
LIN {X 0,Y 530.973,Z 127.349,A -85,B 0,C 180,E1 -4483.07,E2 -4483.07} C_VEL
LIN {X 0,Y 531.02,Z 127.337,A -85,B 0,C 180,E1 -4485.436,E2 -4485.436} C_VEL
LIN {X 0,Y 531.037,Z 127.335,A -85,B 0,C 180,E1 -4488.55,E2 -4488.55} C_VEL
LIN {X 0,Y 531.037,Z 127.332,A -85,B 0,C 180,E1 -4491.629,E2 -4491.629} C_VEL
LIN {X 0,Y 531.119,Z 127.329,A -85,B 0,C 180,E1 -4494.685,E2 -4494.685} C_VEL
LIN {X 0,Y 531.14,Z 127.319,A -85,B 0,C 180,E1 -4497.725,E2 -4497.725} C_VEL
LIN {X 0,Y 531.153,Z 127.325,A -85,B 0,C 180,E1 -4500.758,E2 -4500.758} C_VEL
LIN {X 0,Y 531.102,Z 127.327,A -85,B 0,C 180,E1 -4503.034,E2 -4503.034} C_VEL
LIN {X 0,Y 531.075,Z 127.329,A -85,B 0,C 180,E1 -4506.077,E2 -4506.077} C_VEL
LIN {X 0,Y 531.052,Z 127.337,A -85,B 0,C 180,E1 -4508.37,E2 -4508.37} C_VEL
LIN {X 0,Y 531.052,Z 127.33,A -85,B 0,C 180,E1 -4511.672,E2 -4511.672} C_VEL
LIN {X 0,Y 531.031,Z 127.334,A -85,B 0,C 180,E1 -4514.956,E2 -4514.956} C_VEL
LIN {X 0,Y 530.981,Z 127.34,A -85,B 0,C 180,E1 -4517.723,E2 -4517.723} C_VEL
LIN {X 0,Y 531.024,Z 127.341,A -85,B 0,C 180,E1 -4520.127,E2 -4520.127} C_VEL
LIN {X 0,Y 530.945,Z 127.346,A -85,B 0,C 180,E1 -4522.573,E2 -4522.573} C_VEL
LIN {X 0,Y 530.994,Z 127.337,A -85,B 0,C 180,E1 -4525.058,E2 -4525.058} C_VEL
LIN {X 0,Y 531.008,Z 127.338,A -85,B 0,C 180,E1 -4527.596,E2 -4527.596} C_VEL
LIN {X 0,Y 530.973,Z 127.341,A -85,B 0,C 180,E1 -4530.645,E2 -4530.645} C_VEL
LIN {X 0,Y 530.986,Z 127.345,A -85,B 0,C 180,E1 -4533.773,E2 -4533.773} C_VEL
LIN {X 0,Y 530.954,Z 127.343,A -85,B 0,C 180,E1 -4536.558,E2 -4536.558} C_VEL
LIN {X 0,Y 530.988,Z 127.342,A -85,B 0,C 180,E1 -4539.443,E2 -4539.443} C_VEL
LIN {X 0,Y 530.977,Z 127.34,A -85,B 0,C 180,E1 -4542.457,E2 -4542.457} C_VEL
LIN {X 0,Y 530.96,Z 127.346,A -85,B 0,C 180,E1 -4543.566,E2 -4543.566} C_VEL
LIN {X 0,Y 530.285,Z 127.428,A -85,B 0,C 180,E1 -4544.199,E2 -4544.199} C_VEL
LIN {X 0,Y 527.438,Z 127.783,A -85,B 0,C 180,E1 -4545.228,E2 -4545.228} C_VEL
LIN {X 0,Y 525.036,Z 128.082,A -85,B 0,C 180,E1 -4546.056,E2 -4546.056} C_VEL
LIN {X 0,Y 524.003,Z 128.208,A -85,B 0,C 180,E1 -4546.696,E2 -4546.696} C_VEL
LIN {X 0,Y 523.918,Z 128.219,A -85,B 0,C 180,E1 -4546.912,E2 -4546.912} C_VEL
LIN {X 0,Y 523.948,Z 128.218,A -85,B 0,C 180,E1 -4549.921,E2 -4549.921} C_VEL
LIN {X 0,Y 523.906,Z 128.221,A -85,B 0,C 180,E1 -4552.868,E2 -4552.868} C_VEL
LIN {X 0,Y 523.919,Z 128.223,A -85,B 0,C 180,E1 -4555.709,E2 -4555.709} C_VEL
LIN {X 0,Y 523.918,Z 128.218,A -85,B 0,C 180,E1 -4558.456,E2 -4558.456} C_VEL
LIN {X 0,Y 523.935,Z 128.223,A -85,B 0,C 180,E1 -4561.125,E2 -4561.125} C_VEL
LIN {X 0,Y 523.984,Z 128.211,A -85,B 0,C 180,E1 -4563.98,E2 -4563.98} C_VEL
LIN {X 0,Y 523.924,Z 128.218,A -85,B 0,C 180,E1 -4566.27,E2 -4566.27} C_VEL
LIN {X 0,Y 523.945,Z 128.219,A -85,B 0,C 180,E1 -4568.767,E2 -4568.767} C_VEL
LIN {X 0,Y 523.946,Z 128.222,A -85,B 0,C 180,E1 -4571.221,E2 -4571.221} C_VEL
LIN {X 0,Y 523.929,Z 128.218,A -85,B 0,C 180,E1 -4573.639,E2 -4573.639} C_VEL
LIN {X 0,Y 523.935,Z 128.216,A -85,B 0,C 180,E1 -4576.028,E2 -4576.028} C_VEL
LIN {X 0,Y 524.013,Z 128.209,A -85,B 0,C 180,E1 -4578.394,E2 -4578.394} C_VEL
LIN {X 0,Y 523.988,Z 128.21,A -85,B 0,C 180,E1 -4581.516,E2 -4581.516} C_VEL
LIN {X 0,Y 524.08,Z 128.205,A -85,B 0,C 180,E1 -4584.614,E2 -4584.614} C_VEL
LIN {X 0,Y 524.112,Z 128.196,A -85,B 0,C 180,E1 -4587.695,E2 -4587.695} C_VEL
LIN {X 0,Y 524.119,Z 128.203,A -85,B 0,C 180,E1 -4590.768,E2 -4590.768} C_VEL
LIN {X 0,Y 524.025,Z 128.253,A -85,B 0,C 180,E1 -4591.009,E2 -4591.009} C_VEL
LIN {X 0,Y 524.449,Z 134.796,A -85,B 0,C 180,E1 -4592.304,E2 -4592.304} C_VEL
LIN {X 0,Y 524.231,Z 148.178,A -85,B 0,C 180,E1 -4594.903,E2 -4594.903} C_VEL
LIN {X 0,Y 525.996,Z 158.367,A -85,B 0,C 180,E1 -4595.103,E2 -4595.103} C_VEL
LIN {X 0,Y 525.491,Z 255.253,A -85,B 0,C 180,E1 -4596.455,E2 -4596.455} C_VEL
LIN {X 0,Y 525.327,Z 268.273,A -85,B 0,C 180,E1 -4596.795,E2 -4596.795} C_VEL
LIN {X 0,Y 525.152,Z 280.448,A -85,B 0,C 180,E1 -4597.264,E2 -4597.264} C_VEL
LIN {X 0,Y 524.938,Z 291.065,A -85,B 0,C 180,E1 -4597.808,E2 -4597.808} C_VEL
LIN {X 0,Y 524.682,Z 302.648,A -85,B 0,C 180,E1 -4598.57,E2 -4598.57} C_VEL
LIN {X 0,Y 524.373,Z 313.28,A -85,B 0,C 180,E1 -4599.45,E2 -4599.45} C_VEL
LIN {X 0,Y 524.114,Z 322.864,A -85,B 0,C 180,E1 -4600.43,E2 -4600.43} C_VEL
LIN {X 0,Y 523.888,Z 332.079,A -85,B 0,C 180,E1 -4601.609,E2 -4601.609} C_VEL
LIN {X 0,Y 523.682,Z 339.518,A -85,B 0,C 180,E1 -4602.794,E2 -4602.794} C_VEL
LIN {X 0,Y 523.563,Z 345.476,A -85,B 0,C 180,E1 -4603.982,E2 -4603.982} C_VEL
LIN {X 0,Y 523.485,Z 350.023,A -85,B 0,C 180,E1 -4605.137,E2 -4605.137} C_VEL
LIN {X 0,Y 523.365,Z 353.724,A -85,B 0,C 180,E1 -4606.38,E2 -4606.38} C_VEL
LIN {X 0,Y 523.32,Z 356.147,A -85,B 0,C 180,E1 -4607.541,E2 -4607.541} C_VEL
LIN {X 0,Y 523.305,Z 357.725,A -85,B 0,C 180,E1 -4608.803,E2 -4608.803} C_VEL
LIN {X 0,Y 523.31,Z 358.221,A -85,B 0,C 180,E1 -4609.933,E2 -4609.933} C_VEL
LIN {X 0,Y 523.296,Z 357.751,A -85,B 0,C 180,E1 -4611.261,E2 -4611.261} C_VEL
LIN {X 0,Y 523.338,Z 356.837,A -85,B 0,C 180,E1 -4612.087,E2 -4612.087} C_VEL
LIN {X 0,Y 523.329,Z 355.467,A -85,B 0,C 180,E1 -4612.921,E2 -4612.921} C_VEL
LIN {X 0,Y 523.431,Z 352.757,A -85,B 0,C 180,E1 -4614.074,E2 -4614.074} C_VEL
LIN {X 0,Y 523.512,Z 348.268,A -85,B 0,C 180,E1 -4615.442,E2 -4615.442} C_VEL
LIN {X 0,Y 523.644,Z 342.618,A -85,B 0,C 180,E1 -4616.719,E2 -4616.719} C_VEL
LIN {X 0,Y 523.802,Z 335.293,A -85,B 0,C 180,E1 -4618.009,E2 -4618.009} C_VEL
LIN {X 0,Y 524.032,Z 327.505,A -85,B 0,C 180,E1 -4619.107,E2 -4619.107} C_VEL
LIN {X 0,Y 524.209,Z 319.164,A -85,B 0,C 180,E1 -4620.072,E2 -4620.072} C_VEL
LIN {X 0,Y 524.457,Z 309.221,A -85,B 0,C 180,E1 -4621.006,E2 -4621.006} C_VEL
LIN {X 0,Y 524.75,Z 298.389,A -85,B 0,C 180,E1 -4621.827,E2 -4621.827} C_VEL
LIN {X 0,Y 525.098,Z 286.799,A -85,B 0,C 180,E1 -4622.52,E2 -4622.52} C_VEL
LIN {X 0,Y 525.287,Z 275.131,A -85,B 0,C 180,E1 -4623.053,E2 -4623.053} C_VEL
LIN {X 0,Y 525.449,Z 262.929,A -85,B 0,C 180,E1 -4623.455,E2 -4623.455} C_VEL
LIN {X 0,Y 525.559,Z 249.691,A -85,B 0,C 180,E1 -4623.731,E2 -4623.731} C_VEL
LIN {X 0,Y 525.865,Z 156.461,A -85,B 0,C 180,E1 -4625.02,E2 -4625.02} C_VEL
LIN {X 0,Y 524.25,Z 148.175,A -85,B 0,C 180,E1 -4625.201,E2 -4625.201} C_VEL
LIN {X 0,Y 524.456,Z 133.307,A -85,B 0,C 180,E1 -4628.056,E2 -4628.056} C_VEL
LIN {X 0,Y 523.975,Z 128.22,A -85,B 0,C 180,E1 -4629.08,E2 -4629.08} C_VEL
LIN {X 0,Y 523.899,Z 128.224,A -85,B 0,C 180,E1 -4632.124,E2 -4632.124} C_VEL
LIN {X 0,Y 523.934,Z 128.226,A -85,B 0,C 180,E1 -4635.311,E2 -4635.311} C_VEL
LIN {X 0,Y 523.92,Z 128.224,A -85,B 0,C 180,E1 -4638.695,E2 -4638.695} C_VEL
LIN {X 0,Y 523.912,Z 128.221,A -85,B 0,C 180,E1 -4641.898,E2 -4641.898} C_VEL
LIN {X 0,Y 523.917,Z 128.226,A -85,B 0,C 180,E1 -4644.913,E2 -4644.913} C_VEL
LIN {X 0,Y 523.93,Z 128.219,A -85,B 0,C 180,E1 -4647.681,E2 -4647.681} C_VEL
LIN {X 0,Y 523.93,Z 128.226,A -85,B 0,C 180,E1 -4650.682,E2 -4650.682} C_VEL
LIN {X 0,Y 523.89,Z 128.223,A -85,B 0,C 180,E1 -4653.724,E2 -4653.724} C_VEL
LIN {X 0,Y 523.895,Z 128.227,A -85,B 0,C 180,E1 -4656.269,E2 -4656.269} C_VEL
LIN {X 0,Y 523.898,Z 128.228,A -85,B 0,C 180,E1 -4658.765,E2 -4658.765} C_VEL
LIN {X 0,Y 523.895,Z 128.221,A -85,B 0,C 180,E1 -4661.219,E2 -4661.219} C_VEL
LIN {X 0,Y 523.874,Z 128.225,A -85,B 0,C 180,E1 -4663.637,E2 -4663.637} C_VEL
LIN {X 0,Y 523.891,Z 128.225,A -85,B 0,C 180,E1 -4666.027,E2 -4666.027} C_VEL
LIN {X 0,Y 523.96,Z 128.217,A -85,B 0,C 180,E1 -4668.393,E2 -4668.393} C_VEL
LIN {X 0,Y 523.943,Z 128.217,A -85,B 0,C 180,E1 -4671.515,E2 -4671.515} C_VEL
LIN {X 0,Y 524.027,Z 128.206,A -85,B 0,C 180,E1 -4674.613,E2 -4674.613} C_VEL
LIN {X 0,Y 524.103,Z 128.2,A -85,B 0,C 180,E1 -4677.695,E2 -4677.695} C_VEL
LIN {X 0,Y 524.097,Z 128.203,A -85,B 0,C 180,E1 -4680,E2 -4680} C_VEL
LIN {X 0,Y 524.104,Z 128.194,A -85,B 0,C 180,E1 -4682.306,E2 -4682.306} C_VEL
LIN {X 0,Y 524.002,Z 128.21,A -85,B 0,C 180,E1 -4686.16,E2 -4686.16} C_VEL
LIN {X 0,Y 523.949,Z 128.217,A -85,B 0,C 180,E1 -4689.263,E2 -4689.263} C_VEL
LIN {X 0,Y 524,Z 128.212,A -85,B 0,C 180,E1 -4691.736,E2 -4691.736} C_VEL
LIN {X 0,Y 523.986,Z 128.214,A -85,B 0,C 180,E1 -4695.048,E2 -4695.048} C_VEL
LIN {X 0,Y 523.917,Z 128.218,A -85,B 0,C 180,E1 -4697.971,E2 -4697.971} C_VEL
LIN {X 0,Y 523.96,Z 128.214,A -85,B 0,C 180,E1 -4700.411,E2 -4700.411} C_VEL
LIN {X 0,Y 523.909,Z 128.222,A -85,B 0,C 180,E1 -4702.894,E2 -4702.894} C_VEL
LIN {X 0,Y 523.91,Z 128.222,A -85,B 0,C 180,E1 -4705.421,E2 -4705.421} C_VEL
LIN {X 0,Y 523.911,Z 128.22,A -85,B 0,C 180,E1 -4708.003,E2 -4708.003} C_VEL
LIN {X 0,Y 523.937,Z 128.222,A -85,B 0,C 180,E1 -4710.853,E2 -4710.853} C_VEL
LIN {X 0,Y 523.932,Z 128.216,A -85,B 0,C 180,E1 -4713.73,E2 -4713.73} C_VEL
LIN {X 0,Y 523.905,Z 128.225,A -85,B 0,C 180,E1 -4716.401,E2 -4716.401} C_VEL
LIN {X 0,Y 523.915,Z 128.223,A -85,B 0,C 180,E1 -4719.086,E2 -4719.086} C_VEL
LIN {X 0,Y 523.94,Z 128.22,A -85,B 0,C 180,E1 -4722.12,E2 -4722.12} C_VEL
LIN {X 0,Y 523.943,Z 128.217,A -85,B 0,C 180,E1 -4725.311,E2 -4725.311} C_VEL
LIN {X 0,Y 523.953,Z 128.22,A -85,B 0,C 180,E1 -4728.691,E2 -4728.691} C_VEL
LIN {X 0,Y 523.92,Z 128.22,A -85,B 0,C 180,E1 -4731.081,E2 -4731.081} C_VEL
LIN {X 0,Y 523.898,Z 128.225,A -85,B 0,C 180,E1 -4733.825,E2 -4733.825} C_VEL
LIN {X 0,Y 523.944,Z 128.22,A -85,B 0,C 180,E1 -4736.636,E2 -4736.636} C_VEL
LIN {X 0,Y 523.95,Z 128.218,A -85,B 0,C 180,E1 -4739.355,E2 -4739.355} C_VEL
LIN {X 0,Y 523.975,Z 128.218,A -85,B 0,C 180,E1 -4742.283,E2 -4742.283} C_VEL
LIN {X 0,Y 523.985,Z 128.261,A -85,B 0,C 180,E1 -4745.113,E2 -4745.113} C_VEL
LIN {X 0,Y 525.354,Z 135.815,A -85,B 0,C 180,E1 -4746.339,E2 -4746.339} C_VEL
LIN {X 0,Y 525.103,Z 148.041,A -85,B 0,C 180,E1 -4748.197,E2 -4748.197} C_VEL
LIN {X 0,Y 524.759,Z 162.95,A -85,B 0,C 180,E1 -4750.438,E2 -4750.438} C_VEL
LIN {X 0,Y 524.461,Z 180.553,A -85,B 0,C 180,E1 -4753.055,E2 -4753.055} C_VEL
LIN {X 0,Y 524.256,Z 192.919,A -85,B 0,C 180,E1 -4754.843,E2 -4754.843} C_VEL
LIN {X 0,Y 525.891,Z 204.48,A -85,B 0,C 180,E1 -4755.051,E2 -4755.051} C_VEL
LIN {X 0,Y 525.475,Z 300.933,A -85,B 0,C 180,E1 -4756.39,E2 -4756.39} C_VEL
LIN {X 0,Y 525.237,Z 314.351,A -85,B 0,C 180,E1 -4756.729,E2 -4756.729} C_VEL
LIN {X 0,Y 525.002,Z 327.731,A -85,B 0,C 180,E1 -4757.239,E2 -4757.239} C_VEL
LIN {X 0,Y 524.738,Z 339.098,A -85,B 0,C 180,E1 -4757.831,E2 -4757.831} C_VEL
LIN {X 0,Y 524.441,Z 350.612,A -85,B 0,C 180,E1 -4758.599,E2 -4758.599} C_VEL
LIN {X 0,Y 524.2,Z 361.11,A -85,B 0,C 180,E1 -4759.474,E2 -4759.474} C_VEL
LIN {X 0,Y 523.943,Z 369.693,A -85,B 0,C 180,E1 -4760.347,E2 -4760.347} C_VEL
LIN {X 0,Y 523.738,Z 377.614,A -85,B 0,C 180,E1 -4761.317,E2 -4761.317} C_VEL
LIN {X 0,Y 523.577,Z 385.354,A -85,B 0,C 180,E1 -4762.48,E2 -4762.48} C_VEL
LIN {X 0,Y 523.458,Z 392.488,A -85,B 0,C 180,E1 -4763.834,E2 -4763.834} C_VEL
LIN {X 0,Y 523.383,Z 397.236,A -85,B 0,C 180,E1 -4764.993,E2 -4764.993} C_VEL
LIN {X 0,Y 523.443,Z 400.869,A -85,B 0,C 180,E1 -4766.151,E2 -4766.151} C_VEL
LIN {X 0,Y 523.391,Z 402.74,A -85,B 0,C 180,E1 -4766.921,E2 -4766.921} C_VEL
LIN {X 0,Y 523.337,Z 404.142,A -85,B 0,C 180,E1 -4767.691,E2 -4767.691} C_VEL
LIN {X 0,Y 523.263,Z 405.754,A -85,B 0,C 180,E1 -4769.23,E2 -4769.23} C_VEL
LIN {X 0,Y 523.265,Z 405.974,A -85,B 0,C 180,E1 -4770,E2 -4770} C_VEL
LIN {X 0,Y 523.275,Z 405.151,A -85,B 0,C 180,E1 -4771.539,E2 -4771.539} C_VEL
LIN {X 0,Y 523.337,Z 404.156,A -85,B 0,C 180,E1 -4772.309,E2 -4772.309} C_VEL
LIN {X 0,Y 523.391,Z 402.758,A -85,B 0,C 180,E1 -4773.079,E2 -4773.079} C_VEL
LIN {X 0,Y 523.422,Z 399.814,A -85,B 0,C 180,E1 -4774.235,E2 -4774.235} C_VEL
LIN {X 0,Y 523.455,Z 395.826,A -85,B 0,C 180,E1 -4775.393,E2 -4775.393} C_VEL
LIN {X 0,Y 523.502,Z 389.769,A -85,B 0,C 180,E1 -4776.731,E2 -4776.731} C_VEL
LIN {X 0,Y 523.644,Z 382.988,A -85,B 0,C 180,E1 -4777.907,E2 -4777.907} C_VEL
LIN {X 0,Y 523.819,Z 374.674,A -85,B 0,C 180,E1 -4779.07,E2 -4779.07} C_VEL
LIN {X 0,Y 524.015,Z 366.15,A -85,B 0,C 180,E1 -4780.041,E2 -4780.041} C_VEL
LIN {X 0,Y 524.295,Z 355.622,A -85,B 0,C 180,E1 -4781.012,E2 -4781.012} C_VEL
LIN {X 0,Y 524.614,Z 343.754,A -85,B 0,C 180,E1 -4781.888,E2 -4781.888} C_VEL
LIN {X 0,Y 524.909,Z 331.852,A -85,B 0,C 180,E1 -4782.566,E2 -4782.566} C_VEL
LIN {X 0,Y 525.147,Z 319.45,A -85,B 0,C 180,E1 -4783.101,E2 -4783.101} C_VEL
LIN {X 0,Y 525.384,Z 306.7,A -85,B 0,C 180,E1 -4783.489,E2 -4783.489} C_VEL
LIN {X 0,Y 525.53,Z 291.497,A -85,B 0,C 180,E1 -4783.756,E2 -4783.756} C_VEL
LIN {X 0,Y 525.787,Z 203.286,A -85,B 0,C 180,E1 -4784.97,E2 -4784.97} C_VEL
LIN {X 0,Y 524.233,Z 192.726,A -85,B 0,C 180,E1 -4785.176,E2 -4785.176} C_VEL
LIN {X 0,Y 524.628,Z 173.755,A -85,B 0,C 180,E1 -4787.986,E2 -4787.986} C_VEL
LIN {X 0,Y 525.126,Z 151.065,A -85,B 0,C 180,E1 -4791.389,E2 -4791.389} C_VEL
LIN {X 0,Y 525.409,Z 136.159,A -85,B 0,C 180,E1 -4793.659,E2 -4793.659} C_VEL
LIN {X 0,Y 523.977,Z 128.217,A -85,B 0,C 180,E1 -4794.966,E2 -4794.966} C_VEL
LIN {X 0,Y 523.959,Z 128.222,A -85,B 0,C 180,E1 -4797.999,E2 -4797.999} C_VEL
LIN {X 0,Y 523.946,Z 128.217,A -85,B 0,C 180,E1 -4800.854,E2 -4800.854} C_VEL
LIN {X 0,Y 523.961,Z 128.219,A -85,B 0,C 180,E1 -4803.734,E2 -4803.734} C_VEL
